# B&R Automation Studio project BenchEDM_AS6 (part 4)

#### HA_Matrix.fun - Exported functions and function blocks
```iecst
FUNCTION HA_Matrix_Tran : BOOL
	VAR_INPUT
		pIn : UDINT;
		pOut : UDINT;
	END_VAR
	VAR
		Internal : HA_Matrix_Internal_typ;
	END_VAR
END_FUNCTION

FUNCTION HA_Matrix_SwapR : BOOL
	VAR_INPUT
		Swap1 : DINT;
		Swap2 : DINT;
		pIn : UDINT;
	END_VAR
	VAR
		Internal : HA_Matrix_Internal_typ;
	END_VAR
END_FUNCTION

FUNCTION HA_Matrix_SwapC : BOOL
	VAR_INPUT
		Swap1 : DINT;
		Swap2 : DINT;
		pIn : UDINT;
	END_VAR
	VAR
		Internal : HA_Matrix_Internal_typ;
	END_VAR
END_FUNCTION

FUNCTION HA_Matrix_Sub : BOOL
	VAR_INPUT
		pIn1 : UDINT;
		pIn2 : UDINT;
		pOut : UDINT;
	END_VAR
	VAR
		Internal : HA_Matrix_Internal_typ;
	END_VAR
END_FUNCTION

FUNCTION HA_Matrix_Rref : BOOL
	VAR_INPUT
		pIn : UDINT;
		pOut : UDINT;
	END_VAR
	VAR
		Internal : HA_Matrix_Internal_typ;
	END_VAR
END_FUNCTION

FUNCTION HA_Matrix_Mult : BOOL
	VAR_INPUT
		pIn1 : UDINT;
		pIn2 : UDINT;
		pOut : UDINT;
	END_VAR
	VAR
		Internal : HA_Matrix_Internal_typ;
	END_VAR
END_FUNCTION

FUNCTION HA_Matrix_Inc : BOOL
	VAR_INPUT
		pIn : UDINT;
	END_VAR
	VAR
		Internal : HA_Matrix_Internal_typ;
	END_VAR
END_FUNCTION

FUNCTION HA_Matrix_I : BOOL
	VAR_INPUT
		pIn : UDINT;
	END_VAR
	VAR
		Internal : HA_Matrix_Internal_typ;
	END_VAR
END_FUNCTION

FUNCTION HA_Matrix_Fill : BOOL
	VAR_INPUT
		FillValue : LREAL;
		pIn : UDINT;
	END_VAR
	VAR
		Internal : HA_Matrix_Internal_typ;
	END_VAR
END_FUNCTION

FUNCTION HA_Matrix_Det : LREAL
	VAR_INPUT
		pIn : UDINT;
		pTemp : UDINT;
		pResult : UDINT;
	END_VAR
	VAR
		Internal : HA_Matrix_Internal_typ;
	END_VAR
END_FUNCTION

FUNCTION HA_Matrix_Add : BOOL
	VAR_INPUT
		pIn1 : UDINT;
		pIn2 : UDINT;
		pOut : UDINT;
	END_VAR
	VAR
		Internal : HA_Matrix_Internal_typ;
	END_VAR
END_FUNCTION

FUNCTION HA_Matrix_Cholesky : BOOL
	VAR_INPUT
		pIn : UDINT;
		pOut : UDINT;
	END_VAR
	VAR
		Internal : HA_Matrix_Internal_typ;
	END_VAR
END_FUNCTION

FUNCTION HA_Matrix_CholSolve : BOOL
	VAR_INPUT
		pL : UDINT;
		pB : UDINT;
		pOut : UDINT;
	END_VAR
	VAR
		Internal : HA_Matrix_Internal_typ;
	END_VAR
END_FUNCTION

FUNCTION HA_Matrix_XtX : BOOL
	VAR_INPUT
		pX : UDINT;
		pOut : UDINT;
	END_VAR
	VAR
		Internal : HA_Matrix_Internal_typ;
	END_VAR
END_FUNCTION

FUNCTION HA_Matrix_XtY : BOOL
	VAR_INPUT
		pX : UDINT;
		pY : UDINT;
		pOut : UDINT;
	END_VAR
	VAR
		Internal : HA_Matrix_Internal_typ;
	END_VAR
END_FUNCTION

FUNCTION HA_Matrix_AddRidge : BOOL
	VAR_INPUT
		pInOut : UDINT;
		Lambda : LREAL;
	END_VAR
	VAR
		Internal : HA_Matrix_Internal_typ;
	END_VAR
END_FUNCTION

FUNCTION HA_Matrix_RLS : BOOL
	VAR_INPUT
		pTheta : UDINT;
		pP : UDINT;
		pX : UDINT;
		Y : LREAL;
		Lambda : LREAL;
		pTemp : UDINT;
	END_VAR
	VAR
		Internal : HA_Matrix_Internal_typ;
	END_VAR
END_FUNCTION

FUNCTION HA_Matrix_RLS_Init : BOOL
	VAR_INPUT
		pTheta : UDINT;
		pP : UDINT;
		InitVariance : LREAL;
	END_VAR
	VAR
		Internal : HA_Matrix_Internal_typ;
	END_VAR
END_FUNCTION

FUNCTION HA_Matrix_Predict : BOOL
	VAR_INPUT
		pX : UDINT;
		pBeta : UDINT;
		pOut : UDINT;
	END_VAR
	VAR
		Internal : HA_Matrix_Internal_typ;
	END_VAR
END_FUNCTION

FUNCTION HA_Matrix_BuildLags : BOOL
	VAR_INPUT
		pY_history : UDINT;
		pU_history : UDINT;
		LagOrder : DINT;
		NumOutputs : DINT;
		NumInputs : DINT;
		pOut : UDINT;
	END_VAR
	VAR
		Internal : HA_Matrix_Internal_typ;
	END_VAR
END_FUNCTION

FUNCTION HA_Matrix_RollingUpdate : BOOL
	VAR_INPUT
		pBuffer : UDINT;
		NewValue : LREAL;
	END_VAR
	VAR
		Internal : HA_Matrix_Internal_typ;
	END_VAR
END_FUNCTION

FUNCTION HA_Matrix_RMSE : LREAL
	VAR_INPUT
		pY_true : UDINT;
		pY_pred : UDINT;
	END_VAR
	VAR
		Internal : HA_Matrix_Internal_typ;
	END_VAR
END_FUNCTION

FUNCTION HA_Matrix_Residuals : BOOL
	VAR_INPUT
		pY_true : UDINT;
		pY_pred : UDINT;
		pOut : UDINT;
	END_VAR
	VAR
		Internal : HA_Matrix_Internal_typ;
	END_VAR
END_FUNCTION

FUNCTION HA_Matrix_R2Score : LREAL
	VAR_INPUT
		pY_true : UDINT;
		pY_pred : UDINT;
	END_VAR
	VAR
		Internal : HA_Matrix_Internal_typ;
	END_VAR
END_FUNCTION

FUNCTION HA_Matrix_Standardize : BOOL
	VAR_INPUT
		pX : UDINT;
		pMean : UDINT;
		pStd : UDINT;
		Mode : DINT;
	END_VAR
	VAR
		Internal : HA_Matrix_Internal_typ;
	END_VAR
END_FUNCTION

FUNCTION HA_Matrix_PolyExpand : BOOL
	VAR_INPUT
		pX : UDINT;
		Order : DINT;
		pOut : UDINT;
	END_VAR
	VAR
		Internal : HA_Matrix_Internal_typ;
	END_VAR
END_FUNCTION

FUNCTION HA_Matrix_Diff : BOOL
	VAR_INPUT
		pX : UDINT;
		pOut : UDINT;
	END_VAR
	VAR
		Internal : HA_Matrix_Internal_typ;
	END_VAR
END_FUNCTION

FUNCTION HA_Matrix_AddBias : BOOL
	VAR_INPUT
		pX : UDINT;
		pOut : UDINT;
	END_VAR
	VAR
		Internal : HA_Matrix_Internal_typ;
	END_VAR
END_FUNCTION

FUNCTION HA_Matrix_PredictMultiStep : BOOL
	VAR_INPUT
		pState : UDINT;
		pBeta : UDINT;
		pHistory : UDINT;
		Steps : DINT;
		LagOrder : DINT;
		PolyOrder : DINT;
		UseDerivative : BOOL;
		UseBias : BOOL;
		pOut : UDINT;
		pLagTemp : UDINT;
		pPolyTemp : UDINT;
		pFeatTemp : UDINT;
		pPredTemp : UDINT;
		pWorkState : UDINT;
		pWorkHist : UDINT;
	END_VAR
	VAR
		Internal : HA_Matrix_Internal_typ;
		Success : BOOL;
	END_VAR
END_FUNCTION

FUNCTION HA_Matrix_Ridge_Fit : BOOL
	VAR_INPUT
		pX : UDINT;
		pY : UDINT;
		Lambda : LREAL;
		UseBias : BOOL;
		WarmupSteps : DINT;
		pBeta : UDINT;
		pXtX : UDINT;
		pXtY : UDINT;
		pL : UDINT;
		pXwork : UDINT;
		pYwork : UDINT;
	END_VAR
	VAR
		Internal : HA_Matrix_Internal_typ;
		Success : BOOL;
	END_VAR
END_FUNCTION

FUNCTION HA_Matrix_BuildLagsStride : BOOL
	VAR_INPUT
		pY_history : UDINT;
		pU_history : UDINT;
		LagOrder : DINT;
		NumOutputs : DINT;
		NumInputs : DINT;
		Stride : DINT;
		pOut : UDINT;
	END_VAR
	VAR
		Internal : HA_Matrix_Internal_typ;
	END_VAR
END_FUNCTION

FUNCTION HA_Matrix_InitStateBuffer : BOOL
	VAR_INPUT
		pX : UDINT;
		LagOrder : DINT;
		pState : UDINT;
		pHistory : UDINT;
	END_VAR
	VAR
		Internal : HA_Matrix_Internal_typ;
	END_VAR
END_FUNCTION

FUNCTION HA_Matrix_NGRC_BuildTrainingData : BOOL
	VAR_INPUT
		pX : UDINT;
		LagOrder : DINT;
		PolyOrder : DINT;
		Stride : DINT;
		UseBias : BOOL;
		WarmupSteps : DINT;
		pOut : UDINT;
		pLagWork : UDINT;
		pPolyWork : UDINT;
	END_VAR
	VAR
		Internal : HA_Matrix_Internal_typ;
		Success : BOOL;
	END_VAR
END_FUNCTION

FUNCTION HA_Matrix_NGRC_Fit : BOOL
	VAR_INPUT
		pX : UDINT;
		pY : UDINT;
		LagOrder : DINT;
		PolyOrder : DINT;
		Stride : DINT;
		Lambda : LREAL;
		UseBias : BOOL;
		UseDerivative : BOOL;
		WarmupSteps : DINT;
		pBeta : UDINT;
		pXtX : UDINT;
		pXtY : UDINT;
		pL : UDINT;
		pLagWork : UDINT;
		pPolyWork : UDINT;
		pFeatWork : UDINT;
		pYwork : UDINT;
	END_VAR
	VAR
		Internal : HA_Matrix_Internal_typ;
		Success : BOOL;
	END_VAR
END_FUNCTION

FUNCTION HA_Matrix_NGRC_InitState : BOOL
	VAR_INPUT
		pX : UDINT;
		LagOrder : DINT;
		Stride : DINT;
		pState : UDINT;
		pHistory : UDINT;
	END_VAR
	VAR
		Internal : HA_Matrix_Internal_typ;
	END_VAR
END_FUNCTION

FUNCTION HA_Matrix_NGRC_Predict : BOOL
	VAR_INPUT
		pHistory : UDINT;
		pBeta : UDINT;
		LagOrder : DINT;
		PolyOrder : DINT;
		UseBias : BOOL;
		pOut : UDINT;
		pLagWork : UDINT;
		pPolyWork : UDINT;
		pFeatWork : UDINT;
	END_VAR
	VAR
		Internal : HA_Matrix_Internal_typ;
		Success : BOOL;
	END_VAR
END_FUNCTION

FUNCTION HA_Matrix_NGRC_PredictMultiStep : BOOL
	VAR_INPUT
		pState : UDINT;
		pBeta : UDINT;
		pHistory : UDINT;
		Steps : DINT;
		LagOrder : DINT;
		PolyOrder : DINT;
		Stride : DINT;
		UseBias : BOOL;
		UseDerivative : BOOL;
		pOut : UDINT;
		pLagWork : UDINT;
		pPolyWork : UDINT;
		pFeatWork : UDINT;
		pPredWork : UDINT;
		pWorkState : UDINT;
		pWorkHist : UDINT;
	END_VAR
	VAR
		Internal : HA_Matrix_Internal_typ;
		Success : BOOL;
	END_VAR
END_FUNCTION

FUNCTION_BLOCK FB_NGRC
	VAR_INPUT
		Enable : BOOL;
		Train : BOOL;
		Predict : BOOL;
		PredictSteps : DINT;
		Reset : BOOL;
	END_VAR
	VAR_OUTPUT
		Status : NGRC_Status_enum;
		Error : NGRC_Error_enum;
		Ready : BOOL;
		Busy : BOOL;
		Done : BOOL;
		Stats : NGRC_Stats_typ;
	END_VAR
	VAR_IN_OUT
		Config : NGRC_Config_typ;
		TrainingData : HA_Matrix_Array_typ;
		PredictionOutput : HA_Matrix_Array_typ;
	END_VAR
	VAR
		Internal : NGRC_Internal_typ;
		TrainTrigger : BOOL;
		PredictTrigger : BOOL;
		ResetTrigger : BOOL;
		Success : BOOL;
		StartTime : UDINT;
		NumDims : DINT;
		NumSamples : DINT;
		IsTrained : BOOL;
	END_VAR
END_FUNCTION_BLOCK

FUNCTION_BLOCK FB_NGRC_Online
	VAR_INPUT
		Enable : BOOL;
		NewSample : BOOL;
		PredictNext : BOOL;
		Reset : BOOL;
	END_VAR
	VAR_OUTPUT
		Status : NGRC_Status_enum;
		Error : NGRC_Error_enum;
		Ready : BOOL;
		PredictionValid : BOOL;
	END_VAR
	VAR_IN_OUT
		Config : NGRC_Config_typ;
		CurrentValue : HA_Matrix_Array_typ;
		Prediction : HA_Matrix_Array_typ;
		TrainedModel : FB_NGRC;
	END_VAR
	VAR
		History : HA_Matrix_Array_typ;
		State : HA_Matrix_Array_typ;
		PredWork : HA_Matrix_Array_typ;
		NewSampleTrigger : BOOL;
		PredictTrigger : BOOL;
		Success : BOOL;
		Initialized : BOOL;
		NumDims : DINT;
		i : DINT;
		temp : LREAL;
	END_VAR
END_FUNCTION_BLOCK

FUNCTION_BLOCK FB_NGRC_Simple
	VAR_INPUT
		Execute : BOOL;
		LagOrder : DINT;
		PolyOrder : DINT;
		Stride : DINT;
		Lambda : LREAL;
		PredictSteps : DINT;
	END_VAR
	VAR_OUTPUT
		Done : BOOL;
		Busy : BOOL;
		Error : BOOL;
		ErrorID : NGRC_Error_enum;
	END_VAR
	VAR_IN_OUT
		TrainingData : HA_Matrix_Array_typ;
		Predictions : HA_Matrix_Array_typ;
	END_VAR
	VAR
		Model : FB_NGRC;
		InternalConfig : NGRC_Config_typ;
		InternalTrainData : HA_Matrix_Array_typ;
		InternalPredictions : HA_Matrix_Array_typ;
		ExecuteTrigger : BOOL;
		State : DINT;
	END_VAR
END_FUNCTION_BLOCK

FUNCTION_BLOCK FB_NGRC_Continuous
	VAR_INPUT
		Enable : BOOL;
		Reset : BOOL;
		NewSample : LREAL;
	END_VAR
	VAR_OUTPUT
		PredictedNext : LREAL;
		Predicted5Step : ARRAY[0..4] OF LREAL;
		Status : NGRC_Continuous_Status_typ;
		Metrics : NGRC_Continuous_Metrics_typ;
	END_VAR
	VAR_IN_OUT
		Config : NGRC_Continuous_Config_typ;
	END_VAR
	VAR
		Model_Active : FB_NGRC;
		Model_Training : FB_NGRC;
		Predictor_Online : FB_NGRC_Online;
		DataBuffer : ARRAY[0..499] OF LREAL;
		BufferIndex : DINT := 0;
		BufferFull : BOOL := FALSE;
		TrainingData : HA_Matrix_Array_typ;
		CurrentSample : HA_Matrix_Array_typ;
		PredictionBuffer : HA_Matrix_Array_typ;
		PredictionOutput_Active : HA_Matrix_Array_typ;
		PredictionOutput_Training : HA_Matrix_Array_typ;
		TrainingState : DINT := 0;
		StateFlags : StateFlags_typ;
		ModelSwapReady : BOOL := FALSE;
		SamplesSinceRetrain : DINT := 0;
		RetrainTrigger : BOOL := FALSE;
		PredictionState : DINT := 0;
		MultiStepState : DINT := 0;
		ErrorSum_1Step : LREAL := 0.0;
		ErrorCount_1Step : DINT := 0;
		MaxError_1Step : LREAL := 0.0;
		LastPrediction : LREAL := 0.0;
		ErrorSum_5Step : LREAL := 0.0;
		ErrorCount_5Step : DINT := 0;
		ErrorWindow : ARRAY[0..19] OF LREAL;
		ErrorWindowIndex : DINT := 0;
		PredictionHistory : ARRAY[0..4] OF LREAL;
		PredictionAge : ARRAY[0..4] OF DINT;
		i : DINT;
		j : DINT;
		temp : LREAL;
		CycleCount : DINT := 0;
	END_VAR
END_FUNCTION_BLOCK

FUNCTION_BLOCK FB_NGRC_Continuous_MultiVar
VAR_INPUT
	Enable : BOOL;
	Reset : BOOL;
	NewSample : ARRAY[0..9] OF LREAL;
END_VAR
VAR_OUTPUT
	PredictedNext : ARRAY[0..9] OF LREAL;
	Predicted5Step : ARRAY[0..9, 0..4] OF LREAL;
	Status : NGRC_MultiVar_Status_typ;
	Metrics : NGRC_MultiVar_Metrics_typ;
END_VAR
VAR_IN_OUT
	Config : NGRC_MultiVar_Config_typ;
END_VAR
VAR
	Model_Active : FB_NGRC;
	Model_Training : FB_NGRC;
	Predictor_Online : FB_NGRC_Online;
	DataBuffer : ARRAY[0..4999] OF LREAL;
	BufferIndex : DINT := 0;
	BufferFull : BOOL := FALSE;
	TrainingData : HA_Matrix_Array_typ;
	CurrentSample : HA_Matrix_Array_typ;
	PredictionBuffer : HA_Matrix_Array_typ;
	PredictionOutput_Active : HA_Matrix_Array_typ;
	PredictionOutput_Training : HA_Matrix_Array_typ;
	StateFlags : StateFlags_typ;
	TrainingState : DINT := 0;
	ModelSwapReady : BOOL := FALSE;
	SamplesSinceRetrain : DINT := 0;
	RetrainTrigger : BOOL := FALSE;
	PredictionState : DINT := 0;
	MultiStepState : DINT := 0;
	ErrorSum_1Step : ARRAY[0..9] OF LREAL;
	ErrorCount_1Step : ARRAY[0..9] OF DINT;
	MaxError_1Step : ARRAY[0..9] OF LREAL;
	LastPrediction : ARRAY[0..9] OF LREAL;
	ErrorSum_5Step : ARRAY[0..9] OF LREAL;
	ErrorCount_5Step : ARRAY[0..9] OF DINT;
	ErrorWindow : ARRAY[0..19] OF LREAL;
	ErrorWindowIndex : DINT := 0;
	TotalErrorSum : LREAL := 0.0;
	TotalErrorCount : DINT := 0;
	PredictionHistory : ARRAY[0..9, 0..4] OF LREAL;
	PredictionAge : ARRAY[0..9, 0..4] OF DINT;
	i : DINT;
	j : DINT;
	k : DINT;
	temp : LREAL;
	tempSum : LREAL;
	CycleCount : DINT := 0;
	NumVars : DINT;
	BufferOffset : DINT;
END_VAR
END_FUNCTION_BLOCK
```

#### HA_Matrix_Tran.st
```iecst
(* Transpose *)
FUNCTION HA_Matrix_Tran
	HA_Matrix_Tran		 			:= TRUE;
	brsmemset(ADR(Internal),0,SIZEOF(Internal));
	Internal.sizeArray				:= SIZEOF(LREAL)*(MAX_HA_MATRIX_ARRAY_IDX+1);
	Internal.sizeTotal				:= Internal.sizeArray + SIZEOF(DINT)*2;
	brsmemcpy(ADR(Internal.row1),pIn+Internal.sizeArray,4);
	brsmemcpy(ADR(Internal.col1),pIn+Internal.sizeArray+4,4);
	Internal.row2					:= Internal.col1;
	Internal.col2					:= Internal.row1;
	IF pIn = 0 OR pOut = 0 OR Internal.row1 = 0 OR Internal.col1 = 0 OR Internal.row1*Internal.col1 > MAX_HA_MATRIX_ARRAY_IDX+1 THEN
		HA_Matrix_Tran	 			:= FALSE;
	ELSE
		brsmemset(pOut,0,Internal.sizeTotal);
		brsmemcpy(pOut+Internal.sizeArray,ADR(Internal.row2),4);
		brsmemcpy(pOut+Internal.sizeArray+4,ADR(Internal.col2),4);
		FOR Internal.i1 := 0 TO (Internal.row1*Internal.col1)-1 DO
			brsmemcpy(pOut+(((Internal.i1 MOD Internal.col1)*Internal.row1)+Internal.i1/Internal.col1)*8,pIn+Internal.i1*8,8);
		END_FOR;
	END_IF;
END_FUNCTION
```

#### HA_Matrix_Mult.st
```iecst
(* Multiply *)
FUNCTION HA_Matrix_Mult
	HA_Matrix_Mult 					:= TRUE;
	brsmemset(ADR(Internal),0,SIZEOF(Internal));
	Internal.sizeArray				:= SIZEOF(LREAL)*(MAX_HA_MATRIX_ARRAY_IDX+1);
	Internal.sizeTotal				:= Internal.sizeArray + SIZEOF(DINT)*2;
	brsmemcpy(ADR(Internal.row1),pIn1+Internal.sizeArray,4);
	brsmemcpy(ADR(Internal.col1),pIn1+Internal.sizeArray+4,4);
	brsmemcpy(ADR(Internal.row2),pIn2+Internal.sizeArray,4);
	brsmemcpy(ADR(Internal.col2),pIn2+Internal.sizeArray+4,4);
	IF pIn1 = 0 OR pIn2 = 0 OR pOut = 0 OR Internal.row1 = 0 OR Internal.col1 = 0 OR Internal.row2 = 0 OR Internal.col2 = 0 OR Internal.row1*Internal.col1 > MAX_HA_MATRIX_ARRAY_IDX+1 OR Internal.row2*Internal.col2 > MAX_HA_MATRIX_ARRAY_IDX+1 OR Internal.row1*Internal.col2 > MAX_HA_MATRIX_ARRAY_IDX+1 OR Internal.col1 <> Internal.row2 THEN
		HA_Matrix_Mult	 			:= FALSE;
	ELSE
		brsmemset(pOut,0,Internal.sizeTotal);
		brsmemcpy(pOut+Internal.sizeArray,ADR(Internal.row1),4);
		brsmemcpy(pOut+Internal.sizeArray+4,ADR(Internal.col2),4);
		FOR Internal.i1 := 0 TO Internal.row1-1 DO
		    FOR Internal.i2 := 0 TO Internal.col2-1 DO
		        Internal.result 	:= 0.0;
		        FOR Internal.i3 := 0 TO Internal.col1-1 DO
					brsmemcpy(ADR(Internal.temp1),pIn1+(Internal.i1*Internal.col1+Internal.i3)*8,8);
					brsmemcpy(ADR(Internal.temp2),pIn2+(Internal.i3*Internal.col2+Internal.i2)*8,8);
		            Internal.result := Internal.result + Internal.temp1 * Internal.temp2;
		        END_FOR;
				brsmemcpy(pOut+(Internal.i1*Internal.col2+Internal.i2)*8,ADR(Internal.result),8);
		    END_FOR;
		END_FOR;
	END_IF;
END_FUNCTION
```

#### HA_Matrix_Add.st
```iecst
(* Addition *)
FUNCTION HA_Matrix_Add
	HA_Matrix_Add	 				:= TRUE;
	brsmemset(ADR(Internal),0,SIZEOF(Internal));
	Internal.sizeArray				:= SIZEOF(LREAL)*(MAX_HA_MATRIX_ARRAY_IDX+1);
	Internal.sizeTotal				:= Internal.sizeArray + SIZEOF(DINT)*2;
	brsmemcpy(ADR(Internal.row1),pIn1+Internal.sizeArray,4);
	brsmemcpy(ADR(Internal.col1),pIn1+Internal.sizeArray+4,4);
	brsmemcpy(ADR(Internal.row2),pIn2+Internal.sizeArray,4);
	brsmemcpy(ADR(Internal.col2),pIn2+Internal.sizeArray+4,4);
	IF pIn1 = 0 OR pIn2 = 0 OR pOut = 0 OR Internal.row1 = 0 OR Internal.col1 = 0 OR Internal.row2 = 0 OR Internal.col2 = 0 OR Internal.row1*Internal.col1 > MAX_HA_MATRIX_ARRAY_IDX+1 OR Internal.row2*Internal.col2 > MAX_HA_MATRIX_ARRAY_IDX+1 OR Internal.row1 <> Internal.row2 OR Internal.col1 <> Internal.col2 THEN
		HA_Matrix_Add	 			:= FALSE;
	ELSE
		brsmemset(pOut,0,Internal.sizeTotal);
		brsmemcpy(pOut+Internal.sizeArray,ADR(Internal.row1),4);
		brsmemcpy(pOut+Internal.sizeArray+4,ADR(Internal.col1),4);
		FOR Internal.i1 := 0 TO Internal.row1-1 DO
		    FOR Internal.i2 := 0 TO Internal.col1-1 DO
				brsmemcpy(ADR(Internal.temp1),pIn1+(Internal.i1*Internal.col1+Internal.i2)*8,8);
				brsmemcpy(ADR(Internal.temp2),pIn2+(Internal.i1*Internal.col1+Internal.i2)*8,8);
		        Internal.result 	:= Internal.temp1 + Internal.temp2;
				brsmemcpy(pOut+(Internal.i1*Internal.col1+Internal.i2)*8,ADR(Internal.result),8);
		    END_FOR;
		END_FOR;
	END_IF;
END_FUNCTION
```

#### HA_Matrix_Sub.st
```iecst
(* Subtraction *)
FUNCTION HA_Matrix_Sub
	HA_Matrix_Sub		 			:= TRUE;
	brsmemset(ADR(Internal),0,SIZEOF(Internal));
	Internal.sizeArray				:= SIZEOF(LREAL)*(MAX_HA_MATRIX_ARRAY_IDX+1);
	Internal.sizeTotal				:= Internal.sizeArray + SIZEOF(DINT)*2;
	brsmemcpy(ADR(Internal.row1),pIn1+Internal.sizeArray,4);
	brsmemcpy(ADR(Internal.col1),pIn1+Internal.sizeArray+4,4);
	brsmemcpy(ADR(Internal.row2),pIn2+Internal.sizeArray,4);
	brsmemcpy(ADR(Internal.col2),pIn2+Internal.sizeArray+4,4);
	IF pIn1 = 0 OR pIn2 = 0 OR pOut = 0 OR Internal.row1 = 0 OR Internal.col1 = 0 OR Internal.row2 = 0 OR Internal.col2 = 0 OR Internal.row1*Internal.col1 > MAX_HA_MATRIX_ARRAY_IDX+1 OR Internal.row2*Internal.col2 > MAX_HA_MATRIX_ARRAY_IDX+1 OR Internal.row1 <> Internal.row2 OR Internal.col1 <> Internal.col2 THEN
		HA_Matrix_Sub	 			:= FALSE;
	ELSE
		brsmemset(pOut,0,Internal.sizeTotal);
		brsmemcpy(pOut+Internal.sizeArray,ADR(Internal.row1),4);
		brsmemcpy(pOut+Internal.sizeArray+4,ADR(Internal.col1),4);
		FOR Internal.i1 := 0 TO Internal.row1-1 DO
		    FOR Internal.i2 := 0 TO Internal.col1-1 DO
				brsmemcpy(ADR(Internal.temp1),pIn1+(Internal.i1*Internal.col1+Internal.i2)*8,8);
				brsmemcpy(ADR(Internal.temp2),pIn2+(Internal.i1*Internal.col1+Internal.i2)*8,8);
		        Internal.result 	:= Internal.temp1 - Internal.temp2;
				brsmemcpy(pOut+(Internal.i1*Internal.col1+Internal.i2)*8,ADR(Internal.result),8);
		    END_FOR;
		END_FOR;
	END_IF;
END_FUNCTION
```

#### HA_Matrix_Fill.st
```iecst
(* Fill *)
FUNCTION HA_Matrix_Fill
	HA_Matrix_Fill	 				:= TRUE;
	brsmemset(ADR(Internal),0,SIZEOF(Internal));
	Internal.sizeArray				:= SIZEOF(LREAL)*(MAX_HA_MATRIX_ARRAY_IDX+1);
	Internal.sizeTotal				:= Internal.sizeArray + SIZEOF(DINT)*2;
	brsmemcpy(ADR(Internal.row1),pIn+Internal.sizeArray,4);
	brsmemcpy(ADR(Internal.col1),pIn+Internal.sizeArray+4,4);
	IF pIn = 0 OR Internal.row1 = 0 OR Internal.col1 = 0 OR Internal.row1*Internal.col1 > MAX_HA_MATRIX_ARRAY_IDX+1 THEN
		HA_Matrix_Fill	 			:= FALSE;
	ELSE
		FOR Internal.i1 := 0 TO Internal.row1-1 DO
		    FOR Internal.i2 := 0 TO Internal.col1-1 DO
				brsmemcpy(pIn+(Internal.i1*Internal.col1+Internal.i2)*8,ADR(FillValue),8);
		    END_FOR;
		END_FOR;
	END_IF;
END_FUNCTION
```

#### HA_Matrix_Inc.st
```iecst
(* Fill Incrementing *)
FUNCTION HA_Matrix_Inc
	HA_Matrix_Inc	 				:= TRUE;
	brsmemset(ADR(Internal),0,SIZEOF(Internal));
	Internal.sizeArray				:= SIZEOF(LREAL)*(MAX_HA_MATRIX_ARRAY_IDX+1);
	Internal.sizeTotal				:= Internal.sizeArray + SIZEOF(DINT)*2;
	brsmemcpy(ADR(Internal.row1),pIn+Internal.sizeArray,4);
	brsmemcpy(ADR(Internal.col1),pIn+Internal.sizeArray+4,4);
	IF pIn = 0 OR Internal.row1 = 0 OR Internal.col1 = 0 OR Internal.row1*Internal.col1 > MAX_HA_MATRIX_ARRAY_IDX+1 THEN
		HA_Matrix_Inc	 			:= FALSE;
	ELSE
		FOR Internal.i1 := 0 TO Internal.row1-1 DO
		    FOR Internal.i2 := 0 TO Internal.col1-1 DO
				Internal.temp1 		:= DINT_TO_LREAL(Internal.i1*Internal.col1+Internal.i2);
				brsmemcpy(pIn+(Internal.i1*Internal.col1+Internal.i2)*8,ADR(Internal.temp1),8);
		    END_FOR;
		END_FOR;
	END_IF;
END_FUNCTION
```

#### HA_Matrix_I.st
```iecst
(* Identity *)
FUNCTION HA_Matrix_I
	HA_Matrix_I	 					:= TRUE;
	brsmemset(ADR(Internal),0,SIZEOF(Internal));
	Internal.sizeArray				:= SIZEOF(LREAL)*(MAX_HA_MATRIX_ARRAY_IDX+1);
	Internal.sizeTotal				:= Internal.sizeArray + SIZEOF(DINT)*2;
	brsmemcpy(ADR(Internal.row1),pIn+Internal.sizeArray,4);
	brsmemcpy(ADR(Internal.col1),pIn+Internal.sizeArray+4,4);
	IF pIn = 0 OR Internal.row1 = 0 OR Internal.col1 = 0 OR Internal.row1*Internal.col1 > MAX_HA_MATRIX_ARRAY_IDX+1 OR Internal.row1 <> Internal.col1 THEN
		HA_Matrix_I	 				:= FALSE;
	ELSE
		FOR Internal.i1 := 0 TO Internal.row1-1 DO
		    FOR Internal.i2 := 0 TO Internal.col1-1 DO
				Internal.temp1 		:= 0.0;
				IF Internal.i1 = Internal.i2 THEN
					Internal.temp1 	:= 1.0;
				END_IF;
				brsmemcpy(pIn+(Internal.i1*Internal.row1+Internal.i2)*8,ADR(Internal.temp1),8);
		    END_FOR;
		END_FOR;
	END_IF;
END_FUNCTION
```

#### HA_Matrix_SwapR.st
```iecst
(* Swap Row *)
FUNCTION HA_Matrix_SwapR
	HA_Matrix_SwapR	 				:= TRUE;
	brsmemset(ADR(Internal),0,SIZEOF(Internal));
	Internal.sizeArray				:= SIZEOF(LREAL)*(MAX_HA_MATRIX_ARRAY_IDX+1);
	Internal.sizeTotal				:= Internal.sizeArray + SIZEOF(DINT)*2;
	brsmemcpy(ADR(Internal.row1),pIn+Internal.sizeArray,4);
	brsmemcpy(ADR(Internal.col1),pIn+Internal.sizeArray+4,4);
	IF pIn = 0 OR Internal.row1 = 0 OR Internal.col1 = 0 OR Internal.row1*Internal.col1 > MAX_HA_MATRIX_ARRAY_IDX+1 OR Swap1 = Swap2 OR Internal.row1-1 < Swap1 OR Internal.row1-1 < Swap2 THEN
		HA_Matrix_SwapR	 			:= FALSE;
	ELSE
		FOR Internal.i1 := 0 TO Internal.col1-1 DO
			brsmemcpy(ADR(Internal.temp1),pIn+(Swap1*Internal.col1+Internal.i1)*8,8);
			brsmemcpy(ADR(Internal.temp2),pIn+(Swap2*Internal.col1+Internal.i1)*8,8);
			brsmemcpy(pIn+(Swap1*Internal.col1+Internal.i1)*8,ADR(Internal.temp2),8);
			brsmemcpy(pIn+(Swap2*Internal.col1+Internal.i1)*8,ADR(Internal.temp1),8);
		END_FOR;
	END_IF;
END_FUNCTION
```

#### HA_Matrix_SwapC.st
```iecst
(* Swap Column *)
FUNCTION HA_Matrix_SwapC
	HA_Matrix_SwapC	 				:= TRUE;
	brsmemset(ADR(Internal),0,SIZEOF(Internal));
	Internal.sizeArray				:= SIZEOF(LREAL)*(MAX_HA_MATRIX_ARRAY_IDX+1);
	Internal.sizeTotal				:= Internal.sizeArray + SIZEOF(DINT)*2;
	brsmemcpy(ADR(Internal.row1),pIn+Internal.sizeArray,4);
	brsmemcpy(ADR(Internal.col1),pIn+Internal.sizeArray+4,4);
	IF pIn = 0 OR Internal.row1 = 0 OR Internal.col1 = 0 OR Internal.row1*Internal.col1 > MAX_HA_MATRIX_ARRAY_IDX+1 OR Swap1 = Swap2 OR Internal.col1-1 < Swap1 OR Internal.col1-1 < Swap2 THEN
		HA_Matrix_SwapC	 			:= FALSE;
	ELSE
		FOR Internal.i1 := 0 TO Internal.row1-1 DO
			brsmemcpy(ADR(Internal.temp1),pIn+(Internal.i1*Internal.col1+Swap1)*8,8);
			brsmemcpy(ADR(Internal.temp2),pIn+(Internal.i1*Internal.col1+Swap2)*8,8);
			brsmemcpy(pIn+(Internal.i1*Internal.col1+Swap1)*8,ADR(Internal.temp2),8);
			brsmemcpy(pIn+(Internal.i1*Internal.col1+Swap2)*8,ADR(Internal.temp1),8);
		END_FOR;
	END_IF;
END_FUNCTION
```

#### HA_Matrix_Det.st
```iecst
(* Determinant *)
FUNCTION HA_Matrix_Det

    HA_Matrix_Det := FALSE;
    brsmemset(ADR(Internal),0,SIZEOF(Internal));
    Internal.sizeArray := SIZEOF(LREAL)*(MAX_HA_MATRIX_ARRAY_IDX+1);
    Internal.sizeTotal := Internal.sizeArray + SIZEOF(DINT)*2;
    brsmemcpy(ADR(Internal.row1),pIn+Internal.sizeArray,4);
    brsmemcpy(ADR(Internal.col1),pIn+Internal.sizeArray+4,4);
    IF pIn = 0 OR pTemp = 0 OR pResult = 0 OR Internal.row1 = 0 OR Internal.col1 = 0 OR Internal.row1 <> Internal.col1 OR Internal.row1*Internal.col1 > MAX_HA_MATRIX_ARRAY_IDX+1 THEN
        Internal.result := 0.0;
        brsmemcpy(pResult,ADR(Internal.result),8);
        HA_Matrix_Det := FALSE;
    ELSE
        IF Internal.row1 = 1 THEN
            brsmemcpy(ADR(Internal.result),pIn,8);
            brsmemcpy(pResult,ADR(Internal.result),8);
            HA_Matrix_Det := TRUE;
        ELSIF Internal.row1 = 2 THEN
            brsmemcpy(ADR(Internal.temp1),pIn+0*8,8);
            brsmemcpy(ADR(Internal.temp2),pIn+1*8,8);
            brsmemcpy(ADR(Internal.temp3),pIn+2*8,8);
            brsmemcpy(ADR(Internal.temp4),pIn+3*8,8);
            Internal.result := Internal.temp1*Internal.temp4 - Internal.temp2*Internal.temp3;
            brsmemcpy(pResult,ADR(Internal.result),8);
            HA_Matrix_Det := TRUE;
        ELSE
            Internal.result := 1.0;  (* Use result to track sign *)
            brsmemcpy(pTemp,pIn,Internal.sizeArray);
            brsmemcpy(pTemp+Internal.sizeArray,pIn+Internal.sizeArray,8);
            FOR Internal.i1 := 0 TO Internal.row1-2 DO
                brsmemcpy(ADR(Internal.temp1),pTemp+(Internal.i1*Internal.col1+Internal.i1)*8,8);
                IF ABS(Internal.temp1) < 1.0e-10 THEN
                    FOR Internal.i2 := Internal.i1+1 TO Internal.row1-1 DO
                        brsmemcpy(ADR(Internal.temp1),pTemp+(Internal.i2*Internal.col1+Internal.i1)*8,8);
                        IF ABS(Internal.temp1) > 1.0e-10 THEN
                            FOR Internal.i3 := 0 TO Internal.col1-1 DO
                                brsmemcpy(ADR(Internal.temp2),pTemp+(Internal.i1*Internal.col1+Internal.i3)*8,8);
                                brsmemcpy(ADR(Internal.temp3),pTemp+(Internal.i2*Internal.col1+Internal.i3)*8,8);
                                brsmemcpy(pTemp+(Internal.i1*Internal.col1+Internal.i3)*8,ADR(Internal.temp3),8);
                                brsmemcpy(pTemp+(Internal.i2*Internal.col1+Internal.i3)*8,ADR(Internal.temp2),8);
                            END_FOR;
                            Internal.result := -Internal.result;  (* Negate sign *)
                            EXIT;
                        END_IF;
                    END_FOR;
                END_IF;
                brsmemcpy(ADR(Internal.temp1),pTemp+(Internal.i1*Internal.col1+Internal.i1)*8,8);
                IF ABS(Internal.temp1) < 1.0e-10 THEN
                    Internal.result := 0.0;
                    brsmemcpy(pResult,ADR(Internal.result),8);
                    HA_Matrix_Det := TRUE;  (* Successfully determined matrix is singular *)
                    RETURN;
                END_IF;
                FOR Internal.i2 := Internal.i1+1 TO Internal.row1-1 DO
                    brsmemcpy(ADR(Internal.temp2),pTemp+(Internal.i2*Internal.col1+Internal.i1)*8,8);
                    Internal.temp3 := Internal.temp2/Internal.temp1;
                    FOR Internal.i3 := Internal.i1 TO Internal.col1-1 DO
                        brsmemcpy(ADR(Internal.temp2),pTemp+(Internal.i2*Internal.col1+Internal.i3)*8,8);
                        brsmemcpy(ADR(Internal.temp4),pTemp+(Internal.i1*Internal.col1+Internal.i3)*8,8);
                        Internal.temp2 := Internal.temp2 - Internal.temp3*Internal.temp4;
                        brsmemcpy(pTemp+(Internal.i2*Internal.col1+Internal.i3)*8,ADR(Internal.temp2),8);
                    END_FOR;
                END_FOR;
            END_FOR;
            (* result already contains the sign, now multiply by diagonal elements *)
            FOR Internal.i1 := 0 TO Internal.row1-1 DO
                brsmemcpy(ADR(Internal.temp1),pTemp+(Internal.i1*Internal.col1+Internal.i1)*8,8);
                Internal.result := Internal.result*Internal.temp1;
            END_FOR;
            brsmemcpy(pResult,ADR(Internal.result),8);
            HA_Matrix_Det := TRUE;
        END_IF;
    END_IF;
END_FUNCTION
```

#### HA_Matrix_Rref.st
```iecst
(* Reduced Row Echelon Form *)
FUNCTION HA_Matrix_Rref
	HA_Matrix_Rref		 			:= TRUE;
	brsmemset(ADR(Internal),0,SIZEOF(Internal));
	Internal.sizeArray				:= SIZEOF(LREAL)*(MAX_HA_MATRIX_ARRAY_IDX+1);
	Internal.sizeTotal				:= Internal.sizeArray + SIZEOF(DINT)*2;
	brsmemcpy(ADR(Internal.row1),pIn+Internal.sizeArray,4);
	brsmemcpy(ADR(Internal.col1),pIn+Internal.sizeArray+4,4);
	IF pIn = 0 OR pOut = 0 OR Internal.row1 = 0 OR Internal.col1 = 0 OR Internal.row1*Internal.col1 > MAX_HA_MATRIX_ARRAY_IDX+1 THEN
		HA_Matrix_Rref	 			:= FALSE;
		brsmemset(pOut,0,Internal.sizeTotal);
		Internal.result				:= 0.0;
		IF pOut <> 0 THEN
			brsmemcpy(pOut,ADR(Internal.row1),4);
		END_IF;
	ELSE
	    brsmemcpy(pOut,pIn,Internal.sizeTotal);
        FOR Internal.i1 := 0 TO Internal.row1-1 DO
			brsmemcpy(ADR(Internal.temp1),pOut+(Internal.i1*Internal.col1+Internal.i1)*8,8);
			IF ABS(Internal.temp1) < 1.0e-10 THEN
        		FOR Internal.i2 := Internal.i1+1 TO Internal.row1-1 DO
					brsmemcpy(ADR(Internal.temp1),pOut+(Internal.i2*Internal.col1+Internal.i1)*8,8);
					IF ABS(Internal.temp1) > 1.0e-10 THEN
						FOR Internal.i3 := 0 TO Internal.col1-1 DO
							brsmemcpy(ADR(Internal.temp2),pOut+(Internal.i1*Internal.col1+Internal.i3)*8,8);
							brsmemcpy(ADR(Internal.temp3),pOut+(Internal.i2*Internal.col1+Internal.i3)*8,8);
							brsmemcpy(pOut+(Internal.i1*Internal.col1+Internal.i3)*8,ADR(Internal.temp3),8);
							brsmemcpy(pOut+(Internal.i2*Internal.col1+Internal.i3)*8,ADR(Internal.temp2),8);
						END_FOR;
						EXIT;
					END_IF;
				END_FOR;
			END_IF;
			brsmemcpy(ADR(Internal.temp1),pOut+(Internal.i1*Internal.col1+Internal.i1)*8,8);
			IF ABS(Internal.temp1) > 1.0e-10 THEN
	            FOR Internal.i2 := 0 TO Internal.col1-1 DO
					brsmemcpy(ADR(Internal.temp2),pOut+(Internal.i1*Internal.col1+Internal.i2)*8,8);
	                Internal.temp3 := Internal.temp2 / Internal.temp1;
					brsmemcpy(pOut+(Internal.i1*Internal.col1+Internal.i2)*8,ADR(Internal.temp3),8);
	            END_FOR;
	            FOR Internal.i2 := 0 TO Internal.row1-1 DO
	                IF Internal.i2 <> Internal.i1 THEN
						brsmemcpy(ADR(Internal.temp1),pOut+(Internal.i2*Internal.col1+Internal.i1)*8,8);
	                    FOR Internal.i3 := 0 TO Internal.col1-1 DO
							brsmemcpy(ADR(Internal.temp2),pOut+(Internal.i2*Internal.col1+Internal.i3)*8,8);
							brsmemcpy(ADR(Internal.temp3),pOut+(Internal.i1*Internal.col1+Internal.i3)*8,8);
							Internal.temp4 := Internal.temp2 - Internal.temp1 * Internal.temp3;
							IF ABS(Internal.temp4) < 1.0e-10 THEN
								Internal.temp4 := 0.0;
							END_IF;
							brsmemcpy(pOut+(Internal.i2*Internal.col1+Internal.i3)*8,ADR(Internal.temp4),8);
	                    END_FOR;
	                END_IF;
	            END_FOR;
			END_IF;
        END_FOR;
		Internal.i3 := 0;
        FOR Internal.i1 := 0 TO Internal.row1-1 DO
			Internal.i4 := 0;
	    	FOR Internal.i2 := 0 TO Internal.col1-1 DO
				brsmemcpy(ADR(Internal.temp1),pOut+(Internal.i1*Internal.col1+Internal.i2)*8,8);
				IF ABS(Internal.temp1) > 1.0e-10 THEN
					Internal.i4 := 1;
				END_IF;
			END_FOR;
			IF Internal.i4 = 0 THEN
				Internal.i3 := Internal.i3 + 1;
			END_IF;
        END_FOR;
		IF pOut <> 0 THEN
			brsmemcpy(pOut,ADR(Internal.i3),4);
		END_IF;
	END_IF;
END_FUNCTION
```

#### HA_Matrix_Cholesky.st
```iecst
(* Cholesky Decomposition *)
FUNCTION HA_Matrix_Cholesky
	HA_Matrix_Cholesky	 			:= TRUE;
	brsmemset(ADR(Internal),0,SIZEOF(Internal));
	Internal.sizeArray				:= SIZEOF(LREAL)*(MAX_HA_MATRIX_ARRAY_IDX+1);
	Internal.sizeTotal				:= Internal.sizeArray + SIZEOF(DINT)*2;
	brsmemcpy(ADR(Internal.row1),pIn+Internal.sizeArray,4);
	brsmemcpy(ADR(Internal.col1),pIn+Internal.sizeArray+4,4);
	IF pIn = 0 OR pOut = 0 OR Internal.row1 = 0 OR Internal.col1 = 0 OR Internal.row1 <> Internal.col1 OR Internal.row1*Internal.col1 > MAX_HA_MATRIX_ARRAY_IDX+1 THEN
		HA_Matrix_Cholesky	 		:= FALSE;
	ELSE
		brsmemset(pOut,0,Internal.sizeTotal);
		brsmemcpy(pOut+Internal.sizeArray,ADR(Internal.row1),4);
		brsmemcpy(pOut+Internal.sizeArray+4,ADR(Internal.col1),4);
		FOR Internal.i1 := 0 TO Internal.row1-1 DO
		    FOR Internal.i2 := 0 TO Internal.i1 DO
				Internal.result 	:= 0.0;
		        IF Internal.i1 = Internal.i2 THEN
		            FOR Internal.i3 := 0 TO Internal.i2-1 DO
						brsmemcpy(ADR(Internal.temp1),pOut+(Internal.i1*Internal.col1+Internal.i3)*8,8);
		                Internal.result := Internal.result + Internal.temp1*Internal.temp1;
		            END_FOR;
					brsmemcpy(ADR(Internal.temp1),pIn+(Internal.i1*Internal.col1+Internal.i1)*8,8);
		            Internal.result := Internal.temp1 - Internal.result;
		            IF Internal.result < 1.0e-10 THEN
		                HA_Matrix_Cholesky := FALSE;
		                RETURN;
		            END_IF;
		            Internal.result := SQRT(Internal.result);
					brsmemcpy(pOut+(Internal.i1*Internal.col1+Internal.i1)*8,ADR(Internal.result),8);
		        ELSE
		            FOR Internal.i3 := 0 TO Internal.i2-1 DO
						brsmemcpy(ADR(Internal.temp1),pOut+(Internal.i1*Internal.col1+Internal.i3)*8,8);
						brsmemcpy(ADR(Internal.temp2),pOut+(Internal.i2*Internal.col1+Internal.i3)*8,8);
		                Internal.result := Internal.result + Internal.temp1*Internal.temp2;
		            END_FOR;
					brsmemcpy(ADR(Internal.temp1),pIn+(Internal.i1*Internal.col1+Internal.i2)*8,8);
					brsmemcpy(ADR(Internal.temp2),pOut+(Internal.i2*Internal.col1+Internal.i2)*8,8);
		            Internal.result := (Internal.temp1 - Internal.result)/Internal.temp2;
					brsmemcpy(pOut+(Internal.i1*Internal.col1+Internal.i2)*8,ADR(Internal.result),8);
		        END_IF;
		    END_FOR;
		END_FOR;
	END_IF;
END_FUNCTION
```

#### HA_Matrix_CholSolve.st
```iecst
(* Cholesky Solve *)
FUNCTION HA_Matrix_CholSolve
	HA_Matrix_CholSolve	 			:= TRUE;
	brsmemset(ADR(Internal),0,SIZEOF(Internal));
	Internal.sizeArray				:= SIZEOF(LREAL)*(MAX_HA_MATRIX_ARRAY_IDX+1);
	Internal.sizeTotal				:= Internal.sizeArray + SIZEOF(DINT)*2;
	brsmemcpy(ADR(Internal.row1),pL+Internal.sizeArray,4);
	brsmemcpy(ADR(Internal.col1),pL+Internal.sizeArray+4,4);
	brsmemcpy(ADR(Internal.row2),pB+Internal.sizeArray,4);
	brsmemcpy(ADR(Internal.col2),pB+Internal.sizeArray+4,4);
	IF pL = 0 OR pB = 0 OR pOut = 0 OR Internal.row1 = 0 OR Internal.col1 = 0 OR Internal.row2 = 0 OR Internal.col2 = 0 OR Internal.row1 <> Internal.col1 OR Internal.row1 <> Internal.row2 OR Internal.row1*Internal.col1 > MAX_HA_MATRIX_ARRAY_IDX+1 OR Internal.row2*Internal.col2 > MAX_HA_MATRIX_ARRAY_IDX+1 THEN
		HA_Matrix_CholSolve	 		:= FALSE;
	ELSE
		brsmemset(pOut,0,Internal.sizeTotal);
		brsmemcpy(pOut+Internal.sizeArray,ADR(Internal.row2),4);
		brsmemcpy(pOut+Internal.sizeArray+4,ADR(Internal.col2),4);
		FOR Internal.i3 := 0 TO Internal.col2-1 DO
		    FOR Internal.i1 := 0 TO Internal.row1-1 DO
				brsmemcpy(ADR(Internal.result),pB+(Internal.i1*Internal.col2+Internal.i3)*8,8);
		        FOR Internal.i2 := 0 TO Internal.i1-1 DO
					brsmemcpy(ADR(Internal.temp1),pL+(Internal.i1*Internal.col1+Internal.i2)*8,8);
					brsmemcpy(ADR(Internal.temp2),pOut+(Internal.i2*Internal.col2+Internal.i3)*8,8);
		            Internal.result := Internal.result - Internal.temp1*Internal.temp2;
		        END_FOR;
				brsmemcpy(ADR(Internal.temp1),pL+(Internal.i1*Internal.col1+Internal.i1)*8,8);
		        Internal.result 	:= Internal.result/Internal.temp1;
				brsmemcpy(pOut+(Internal.i1*Internal.col2+Internal.i3)*8,ADR(Internal.result),8);
		    END_FOR;
		    FOR Internal.i1 := Internal.row1-1 TO 0 BY -1 DO
				brsmemcpy(ADR(Internal.result),pOut+(Internal.i1*Internal.col2+Internal.i3)*8,8);
		        FOR Internal.i2 := Internal.i1+1 TO Internal.row1-1 DO
					brsmemcpy(ADR(Internal.temp1),pL+(Internal.i2*Internal.col1+Internal.i1)*8,8);
					brsmemcpy(ADR(Internal.temp2),pOut+(Internal.i2*Internal.col2+Internal.i3)*8,8);
		            Internal.result := Internal.result - Internal.temp1*Internal.temp2;
		        END_FOR;
				brsmemcpy(ADR(Internal.temp1),pL+(Internal.i1*Internal.col1+Internal.i1)*8,8);
		        Internal.result 	:= Internal.result/Internal.temp1;
				brsmemcpy(pOut+(Internal.i1*Internal.col2+Internal.i3)*8,ADR(Internal.result),8);
		    END_FOR;
		END_FOR;
	END_IF;
END_FUNCTION
```

#### HA_Matrix_RLS.st
```iecst
(* Recursive Least Squares Update *)
FUNCTION HA_Matrix_RLS
	HA_Matrix_RLS	 				:= TRUE;
	brsmemset(ADR(Internal),0,SIZEOF(Internal));
	Internal.sizeArray				:= SIZEOF(LREAL)*(MAX_HA_MATRIX_ARRAY_IDX+1);
	Internal.sizeTotal				:= Internal.sizeArray + SIZEOF(DINT)*2;
	brsmemcpy(ADR(Internal.row1),pTheta+Internal.sizeArray,4);
	brsmemcpy(ADR(Internal.col1),pTheta+Internal.sizeArray+4,4);
	brsmemcpy(ADR(Internal.row2),pP+Internal.sizeArray,4);
	brsmemcpy(ADR(Internal.col2),pP+Internal.sizeArray+4,4);
	brsmemcpy(ADR(Internal.row3),pX+Internal.sizeArray,4);
	brsmemcpy(ADR(Internal.col3),pX+Internal.sizeArray+4,4);
	IF pTheta = 0 OR pP = 0 OR pX = 0 OR Internal.row1 = 0 OR Internal.col1 = 0 OR Internal.row2 = 0 OR Internal.col2 = 0 OR Internal.row3 = 0 OR Internal.col3 = 0 OR Internal.col1 <> 1 OR Internal.row2 <> Internal.col2 OR Internal.row1 <> Internal.row2 OR Internal.row3 <> Internal.row1 OR Internal.col3 <> 1 OR Internal.row1*Internal.col1 > MAX_HA_MATRIX_ARRAY_IDX+1 OR Internal.row2*Internal.col2 > MAX_HA_MATRIX_ARRAY_IDX+1 OR Lambda <= 0.0 OR Lambda > 1.0 THEN
		HA_Matrix_RLS	 			:= FALSE;
	ELSE
		Internal.temp1 				:= 0.0;
		FOR Internal.i1 := 0 TO Internal.row1-1 DO
			Internal.temp2 			:= 0.0;
		    FOR Internal.i2 := 0 TO Internal.row2-1 DO
				brsmemcpy(ADR(Internal.temp3),pP+(Internal.i1*Internal.col2+Internal.i2)*8,8);
				brsmemcpy(ADR(Internal.temp4),pX+(Internal.i2*Internal.col3)*8,8);
		        Internal.temp2 		:= Internal.temp2 + Internal.temp3*Internal.temp4;
		    END_FOR;
			brsmemcpy(pTemp+(Internal.i1*1)*8,ADR(Internal.temp2),8);
			brsmemcpy(ADR(Internal.temp3),pX+(Internal.i1*Internal.col3)*8,8);
			Internal.temp1 			:= Internal.temp1 + Internal.temp3*Internal.temp2;
		END_FOR;
		Internal.temp1 				:= Lambda + Internal.temp1;
		IF ABS(Internal.temp1) < 1.0e-10 THEN
		    HA_Matrix_RLS	 		:= FALSE;
		    RETURN;
		END_IF;
		Internal.result 			:= 0.0;
		FOR Internal.i1 := 0 TO Internal.row1-1 DO
			brsmemcpy(ADR(Internal.temp2),pX+(Internal.i1*Internal.col3)*8,8);
			brsmemcpy(ADR(Internal.temp3),pTheta+(Internal.i1*Internal.col1)*8,8);
		    Internal.result 		:= Internal.result + Internal.temp2*Internal.temp3;
		END_FOR;
		Internal.result 			:= Y - Internal.result;
		FOR Internal.i1 := 0 TO Internal.row1-1 DO
			brsmemcpy(ADR(Internal.temp2),pTemp+(Internal.i1*1)*8,8);
		    Internal.temp3 			:= Internal.temp2/Internal.temp1;
			brsmemcpy(ADR(Internal.temp4),pTheta+(Internal.i1*Internal.col1)*8,8);
			Internal.temp4 			:= Internal.temp4 + Internal.temp3*Internal.result;
			brsmemcpy(pTheta+(Internal.i1*Internal.col1)*8,ADR(Internal.temp4),8);
		END_FOR;
		FOR Internal.i1 := 0 TO Internal.row2-1 DO
		    FOR Internal.i2 := 0 TO Internal.col2-1 DO
				Internal.temp2 		:= 0.0;
		        FOR Internal.i3 := 0 TO Internal.row2-1 DO
					brsmemcpy(ADR(Internal.temp3),pTemp+(Internal.i1*1)*8,8);
					brsmemcpy(ADR(Internal.temp4),pX+(Internal.i3*Internal.col3)*8,8);
					brsmemcpy(ADR(Internal.temp5),pP+(Internal.i3*Internal.col2+Internal.i2)*8,8);
		            Internal.temp2 	:= Internal.temp2 + Internal.temp3*Internal.temp4*Internal.temp5;
		        END_FOR;
				brsmemcpy(ADR(Internal.temp3),pP+(Internal.i1*Internal.col2+Internal.i2)*8,8);
		        Internal.result 	:= (Internal.temp3 - Internal.temp2/Internal.temp1)/Lambda;
				brsmemcpy(pP+(Internal.i1*Internal.col2+Internal.i2)*8,ADR(Internal.result),8);
		    END_FOR;
		END_FOR;
	END_IF;
END_FUNCTION
```

#### HA_Matrix_XtX.st
```iecst
(* Normal Equation X'X *)
FUNCTION HA_Matrix_XtX
	HA_Matrix_XtX	 				:= TRUE;
	brsmemset(ADR(Internal),0,SIZEOF(Internal));
	Internal.sizeArray				:= SIZEOF(LREAL)*(MAX_HA_MATRIX_ARRAY_IDX+1);
	Internal.sizeTotal				:= Internal.sizeArray + SIZEOF(DINT)*2;
	brsmemcpy(ADR(Internal.row1),pX+Internal.sizeArray,4);
	brsmemcpy(ADR(Internal.col1),pX+Internal.sizeArray+4,4);
	Internal.row2					:= Internal.col1;
	Internal.col2					:= Internal.col1;
	IF pX = 0 OR pOut = 0 OR Internal.row1 = 0 OR Internal.col1 = 0 OR Internal.row1*Internal.col1 > MAX_HA_MATRIX_ARRAY_IDX+1 OR Internal.row2*Internal.col2 > MAX_HA_MATRIX_ARRAY_IDX+1 THEN
		HA_Matrix_XtX	 			:= FALSE;
	ELSE
		brsmemset(pOut,0,Internal.sizeTotal);
		brsmemcpy(pOut+Internal.sizeArray,ADR(Internal.row2),4);
		brsmemcpy(pOut+Internal.sizeArray+4,ADR(Internal.col2),4);
		FOR Internal.i1 := 0 TO Internal.col1-1 DO
		    FOR Internal.i2 := 0 TO Internal.col1-1 DO
		        Internal.result 	:= 0.0;
		        FOR Internal.i3 := 0 TO Internal.row1-1 DO
					brsmemcpy(ADR(Internal.temp1),pX+(Internal.i3*Internal.col1+Internal.i1)*8,8);
					brsmemcpy(ADR(Internal.temp2),pX+(Internal.i3*Internal.col1+Internal.i2)*8,8);
		            Internal.result := Internal.result + Internal.temp1*Internal.temp2;
		        END_FOR;
				brsmemcpy(pOut+(Internal.i1*Internal.col2+Internal.i2)*8,ADR(Internal.result),8);
		    END_FOR;
		END_FOR;
	END_IF;
END_FUNCTION
```

#### HA_Matrix_XtY.st
```iecst
(* Normal Equation X'Y *)
FUNCTION HA_Matrix_XtY
	HA_Matrix_XtY	 				:= TRUE;
	brsmemset(ADR(Internal),0,SIZEOF(Internal));
	Internal.sizeArray				:= SIZEOF(LREAL)*(MAX_HA_MATRIX_ARRAY_IDX+1);
	Internal.sizeTotal				:= Internal.sizeArray + SIZEOF(DINT)*2;
	brsmemcpy(ADR(Internal.row1),pX+Internal.sizeArray,4);
	brsmemcpy(ADR(Internal.col1),pX+Internal.sizeArray+4,4);
	brsmemcpy(ADR(Internal.row2),pY+Internal.sizeArray,4);
	brsmemcpy(ADR(Internal.col2),pY+Internal.sizeArray+4,4);
	Internal.row3					:= Internal.col1;
	Internal.col3					:= Internal.col2;
	IF pX = 0 OR pY = 0 OR pOut = 0 OR Internal.row1 = 0 OR Internal.col1 = 0 OR Internal.row2 = 0 OR Internal.col2 = 0 OR Internal.row1 <> Internal.row2 OR Internal.row1*Internal.col1 > MAX_HA_MATRIX_ARRAY_IDX+1 OR Internal.row2*Internal.col2 > MAX_HA_MATRIX_ARRAY_IDX+1 OR Internal.row3*Internal.col3 > MAX_HA_MATRIX_ARRAY_IDX+1 THEN
		HA_Matrix_XtY	 			:= FALSE;
	ELSE
		brsmemset(pOut,0,Internal.sizeTotal);
		brsmemcpy(pOut+Internal.sizeArray,ADR(Internal.row3),4);
		brsmemcpy(pOut+Internal.sizeArray+4,ADR(Internal.col3),4);
		FOR Internal.i1 := 0 TO Internal.col1-1 DO
		    FOR Internal.i2 := 0 TO Internal.col2-1 DO
		        Internal.result 	:= 0.0;
		        FOR Internal.i3 := 0 TO Internal.row1-1 DO
					brsmemcpy(ADR(Internal.temp1),pX+(Internal.i3*Internal.col1+Internal.i1)*8,8);
					brsmemcpy(ADR(Internal.temp2),pY+(Internal.i3*Internal.col2+Internal.i2)*8,8);
		            Internal.result := Internal.result + Internal.temp1*Internal.temp2;
		        END_FOR;
				brsmemcpy(pOut+(Internal.i1*Internal.col3+Internal.i2)*8,ADR(Internal.result),8);
		    END_FOR;
		END_FOR;
	END_IF;
END_FUNCTION
```

#### HA_Matrix_AddRidge.st
```iecst
(* Add Ridge Penalty *)
FUNCTION HA_Matrix_AddRidge
	HA_Matrix_AddRidge	 			:= TRUE;
	brsmemset(ADR(Internal),0,SIZEOF(Internal));
	Internal.sizeArray				:= SIZEOF(LREAL)*(MAX_HA_MATRIX_ARRAY_IDX+1);
	Internal.sizeTotal				:= Internal.sizeArray + SIZEOF(DINT)*2;
	brsmemcpy(ADR(Internal.row1),pInOut+Internal.sizeArray,4);
	brsmemcpy(ADR(Internal.col1),pInOut+Internal.sizeArray+4,4);
	IF pInOut = 0 OR Internal.row1 = 0 OR Internal.col1 = 0 OR Internal.row1 <> Internal.col1 OR Internal.row1*Internal.col1 > MAX_HA_MATRIX_ARRAY_IDX+1 OR Lambda < 0.0 THEN
		HA_Matrix_AddRidge	 		:= FALSE;
	ELSE
		FOR Internal.i1 := 0 TO Internal.row1-1 DO
			brsmemcpy(ADR(Internal.temp1),pInOut+(Internal.i1*Internal.col1+Internal.i1)*8,8);
		    Internal.temp1 			:= Internal.temp1 + Lambda;
			brsmemcpy(pInOut+(Internal.i1*Internal.col1+Internal.i1)*8,ADR(Internal.temp1),8);
		END_FOR;
	END_IF;
END_FUNCTION
```

#### HA_Matrix_RLS_Init.st
```iecst
(* Initialize RLS *)
FUNCTION HA_Matrix_RLS_Init
	HA_Matrix_RLS_Init	 			:= TRUE;
	brsmemset(ADR(Internal),0,SIZEOF(Internal));
	Internal.sizeArray				:= SIZEOF(LREAL)*(MAX_HA_MATRIX_ARRAY_IDX+1);
	Internal.sizeTotal				:= Internal.sizeArray + SIZEOF(DINT)*2;
	brsmemcpy(ADR(Internal.row1),pTheta+Internal.sizeArray,4);
	brsmemcpy(ADR(Internal.col1),pTheta+Internal.sizeArray+4,4);
	brsmemcpy(ADR(Internal.row2),pP+Internal.sizeArray,4);
	brsmemcpy(ADR(Internal.col2),pP+Internal.sizeArray+4,4);
	IF pTheta = 0 OR pP = 0 OR Internal.row1 = 0 OR Internal.col1 = 0 OR Internal.row2 = 0 OR Internal.col2 = 0 OR Internal.col1 <> 1 OR Internal.row2 <> Internal.col2 OR Internal.row1 <> Internal.row2 OR Internal.row1*Internal.col1 > MAX_HA_MATRIX_ARRAY_IDX+1 OR Internal.row2*Internal.col2 > MAX_HA_MATRIX_ARRAY_IDX+1 OR InitVariance <= 0.0 THEN
		HA_Matrix_RLS_Init	 		:= FALSE;
	ELSE
		FOR Internal.i1 := 0 TO Internal.row1-1 DO
			Internal.temp1 			:= 0.0;
			brsmemcpy(pTheta+(Internal.i1*Internal.col1)*8,ADR(Internal.temp1),8);
		END_FOR;
		FOR Internal.i1 := 0 TO Internal.row2-1 DO
		    FOR Internal.i2 := 0 TO Internal.col2-1 DO
				Internal.temp1 		:= 0.0;
				IF Internal.i1 = Internal.i2 THEN
					Internal.temp1 	:= InitVariance;
				END_IF;
				brsmemcpy(pP+(Internal.i1*Internal.col2+Internal.i2)*8,ADR(Internal.temp1),8);
		    END_FOR;
		END_FOR;
	END_IF;
END_FUNCTION
```

#### HA_Matrix_BuildLags.st
```iecst
(* Build Lag Matrix *)
FUNCTION HA_Matrix_BuildLags
	HA_Matrix_BuildLags	 			:= TRUE;
	brsmemset(ADR(Internal),0,SIZEOF(Internal));
	Internal.sizeArray				:= SIZEOF(LREAL)*(MAX_HA_MATRIX_ARRAY_IDX+1);
	Internal.sizeTotal				:= Internal.sizeArray + SIZEOF(DINT)*2;
	brsmemcpy(ADR(Internal.row1),pY_history+Internal.sizeArray,4);
	brsmemcpy(ADR(Internal.col1),pY_history+Internal.sizeArray+4,4);
	IF pU_history <> 0 THEN
		brsmemcpy(ADR(Internal.row2),pU_history+Internal.sizeArray,4);
		brsmemcpy(ADR(Internal.col2),pU_history+Internal.sizeArray+4,4);
	ELSE
		Internal.row2 				:= 0;
		Internal.col2 				:= 0;
	END_IF;
	Internal.row3					:= NumOutputs*LagOrder + NumInputs*LagOrder;
	Internal.col3					:= 1;
	IF pY_history = 0 OR pOut = 0 OR LagOrder = 0 OR NumOutputs = 0 OR Internal.row1 = 0 OR Internal.col1 = 0 OR Internal.row1 < NumOutputs*LagOrder OR Internal.col1 <> 1 OR Internal.row3*Internal.col3 > MAX_HA_MATRIX_ARRAY_IDX+1 THEN
		HA_Matrix_BuildLags	 		:= FALSE;
	ELSE
		IF pU_history <> 0 THEN
			IF NumInputs = 0 OR Internal.row2 = 0 OR Internal.col2 = 0 OR Internal.row2 < NumInputs*LagOrder OR Internal.col2 <> 1 THEN
				HA_Matrix_BuildLags	 := FALSE;
				RETURN;
			END_IF;
		END_IF;
		brsmemset(pOut,0,Internal.sizeTotal);
		brsmemcpy(pOut+Internal.sizeArray,ADR(Internal.row3),4);
		brsmemcpy(pOut+Internal.sizeArray+4,ADR(Internal.col3),4);
		Internal.i4 				:= 0;
		FOR Internal.i1 := 0 TO LagOrder-1 DO
		    FOR Internal.i2 := 0 TO NumOutputs-1 DO
				brsmemcpy(ADR(Internal.temp1),pY_history+(Internal.i1*NumOutputs+Internal.i2)*8,8);
				brsmemcpy(pOut+Internal.i4*8,ADR(Internal.temp1),8);
				Internal.i4 			:= Internal.i4 + 1;
		    END_FOR;
		END_FOR;
		IF pU_history <> 0 AND NumInputs > 0 THEN
			FOR Internal.i1 := 0 TO LagOrder-1 DO
			    FOR Internal.i2 := 0 TO NumInputs-1 DO
					brsmemcpy(ADR(Internal.temp1),pU_history+(Internal.i1*NumInputs+Internal.i2)*8,8);
					brsmemcpy(pOut+Internal.i4*8,ADR(Internal.temp1),8);
					Internal.i4 		:= Internal.i4 + 1;
			    END_FOR;
			END_FOR;
		END_IF;
	END_IF;
END_FUNCTION
```

#### HA_Matrix_RollingUpdate.st
```iecst
(* Rolling Buffer Update *)
FUNCTION HA_Matrix_RollingUpdate
	HA_Matrix_RollingUpdate	 		:= TRUE;
	brsmemset(ADR(Internal),0,SIZEOF(Internal));
	Internal.sizeArray				:= SIZEOF(LREAL)*(MAX_HA_MATRIX_ARRAY_IDX+1);
	Internal.sizeTotal				:= Internal.sizeArray + SIZEOF(DINT)*2;
	brsmemcpy(ADR(Internal.row1),pBuffer+Internal.sizeArray,4);
	brsmemcpy(ADR(Internal.col1),pBuffer+Internal.sizeArray+4,4);
	IF pBuffer = 0 OR Internal.row1 = 0 OR Internal.col1 = 0 OR Internal.row1*Internal.col1 > MAX_HA_MATRIX_ARRAY_IDX+1 THEN
		HA_Matrix_RollingUpdate	 	:= FALSE;
	ELSE
		FOR Internal.i1 := Internal.row1*Internal.col1-1 TO 1 BY -1 DO
			brsmemcpy(ADR(Internal.temp1),pBuffer+(Internal.i1-1)*8,8);
			brsmemcpy(pBuffer+Internal.i1*8,ADR(Internal.temp1),8);
		END_FOR;
		brsmemcpy(pBuffer,ADR(NewValue),8);
	END_IF;
END_FUNCTION
```

#### HA_Matrix_Predict.st
```iecst
(* Predict *)
FUNCTION HA_Matrix_Predict
	HA_Matrix_Predict	 			:= TRUE;
	brsmemset(ADR(Internal),0,SIZEOF(Internal));
	Internal.sizeArray				:= SIZEOF(LREAL)*(MAX_HA_MATRIX_ARRAY_IDX+1);
	Internal.sizeTotal				:= Internal.sizeArray + SIZEOF(DINT)*2;
	brsmemcpy(ADR(Internal.row1),pX+Internal.sizeArray,4);
	brsmemcpy(ADR(Internal.col1),pX+Internal.sizeArray+4,4);
	brsmemcpy(ADR(Internal.row2),pBeta+Internal.sizeArray,4);
	brsmemcpy(ADR(Internal.col2),pBeta+Internal.sizeArray+4,4);
	Internal.row3					:= Internal.row1;
	Internal.col3					:= Internal.col2;
	IF pX = 0 OR pBeta = 0 OR pOut = 0 OR Internal.row1 = 0 OR Internal.col1 = 0 OR Internal.row2 = 0 OR Internal.col2 = 0 OR Internal.col1 <> Internal.row2 OR Internal.row1*Internal.col1 > MAX_HA_MATRIX_ARRAY_IDX+1 OR Internal.row2*Internal.col2 > MAX_HA_MATRIX_ARRAY_IDX+1 OR Internal.row3*Internal.col3 > MAX_HA_MATRIX_ARRAY_IDX+1 THEN
		HA_Matrix_Predict	 		:= FALSE;
	ELSE
		brsmemset(pOut,0,Internal.sizeTotal);
		brsmemcpy(pOut+Internal.sizeArray,ADR(Internal.row3),4);
		brsmemcpy(pOut+Internal.sizeArray+4,ADR(Internal.col3),4);
		FOR Internal.i1 := 0 TO Internal.row1-1 DO
		    FOR Internal.i2 := 0 TO Internal.col2-1 DO
		        Internal.result 	:= 0.0;
		        FOR Internal.i3 := 0 TO Internal.col1-1 DO
					brsmemcpy(ADR(Internal.temp1),pX+(Internal.i1*Internal.col1+Internal.i3)*8,8);
					brsmemcpy(ADR(Internal.temp2),pBeta+(Internal.i3*Internal.col2+Internal.i2)*8,8);
		            Internal.result := Internal.result + Internal.temp1*Internal.temp2;
		        END_FOR;
				brsmemcpy(pOut+(Internal.i1*Internal.col3+Internal.i2)*8,ADR(Internal.result),8);
		    END_FOR;
		END_FOR;
	END_IF;
END_FUNCTION
```

#### HA_Matrix_RMSE.st
```iecst
(* Root Mean Square Error *)
FUNCTION HA_Matrix_RMSE
	HA_Matrix_RMSE	 				:= 0.0;
	brsmemset(ADR(Internal),0,SIZEOF(Internal));
	Internal.sizeArray				:= SIZEOF(LREAL)*(MAX_HA_MATRIX_ARRAY_IDX+1);
	Internal.sizeTotal				:= Internal.sizeArray + SIZEOF(DINT)*2;
	brsmemcpy(ADR(Internal.row1),pY_true+Internal.sizeArray,4);
	brsmemcpy(ADR(Internal.col1),pY_true+Internal.sizeArray+4,4);
	brsmemcpy(ADR(Internal.row2),pY_pred+Internal.sizeArray,4);
	brsmemcpy(ADR(Internal.col2),pY_pred+Internal.sizeArray+4,4);
	IF pY_true = 0 OR pY_pred = 0 OR Internal.row1 = 0 OR Internal.col1 = 0 OR Internal.row2 = 0 OR Internal.col2 = 0 OR Internal.row1 <> Internal.row2 OR Internal.col1 <> Internal.col2 OR Internal.row1*Internal.col1 > MAX_HA_MATRIX_ARRAY_IDX+1 THEN
		HA_Matrix_RMSE	 			:= 0.0;
	ELSE
		Internal.result 			:= 0.0;
		FOR Internal.i1 := 0 TO Internal.row1-1 DO
		    FOR Internal.i2 := 0 TO Internal.col1-1 DO
				brsmemcpy(ADR(Internal.temp1),pY_true+(Internal.i1*Internal.col1+Internal.i2)*8,8);
				brsmemcpy(ADR(Internal.temp2),pY_pred+(Internal.i1*Internal.col1+Internal.i2)*8,8);
		        Internal.temp3 		:= Internal.temp1 - Internal.temp2;
		        Internal.result 	:= Internal.result + Internal.temp3*Internal.temp3;
		    END_FOR;
		END_FOR;
		Internal.result 			:= Internal.result/DINT_TO_LREAL(Internal.row1*Internal.col1);
		HA_Matrix_RMSE	 			:= SQRT(Internal.result);
	END_IF;
END_FUNCTION
```

#### HA_Matrix_Residuals.st
```iecst
(* Residuals *)
FUNCTION HA_Matrix_Residuals
	HA_Matrix_Residuals	 			:= TRUE;
	brsmemset(ADR(Internal),0,SIZEOF(Internal));
	Internal.sizeArray				:= SIZEOF(LREAL)*(MAX_HA_MATRIX_ARRAY_IDX+1);
	Internal.sizeTotal				:= Internal.sizeArray + SIZEOF(DINT)*2;
	brsmemcpy(ADR(Internal.row1),pY_true+Internal.sizeArray,4);
	brsmemcpy(ADR(Internal.col1),pY_true+Internal.sizeArray+4,4);
	brsmemcpy(ADR(Internal.row2),pY_pred+Internal.sizeArray,4);
	brsmemcpy(ADR(Internal.col2),pY_pred+Internal.sizeArray+4,4);
	IF pY_true = 0 OR pY_pred = 0 OR pOut = 0 OR Internal.row1 = 0 OR Internal.col1 = 0 OR Internal.row2 = 0 OR Internal.col2 = 0 OR Internal.row1*Internal.col1 > MAX_HA_MATRIX_ARRAY_IDX+1 OR Internal.row2*Internal.col2 > MAX_HA_MATRIX_ARRAY_IDX+1 OR Internal.row1 <> Internal.row2 OR Internal.col1 <> Internal.col2 THEN
		HA_Matrix_Residuals	 		:= FALSE;
	ELSE
		brsmemset(pOut,0,Internal.sizeTotal);
		brsmemcpy(pOut+Internal.sizeArray,ADR(Internal.row1),4);
		brsmemcpy(pOut+Internal.sizeArray+4,ADR(Internal.col1),4);
		FOR Internal.i1 := 0 TO Internal.row1-1 DO
		    FOR Internal.i2 := 0 TO Internal.col1-1 DO
				brsmemcpy(ADR(Internal.temp1),pY_true+(Internal.i1*Internal.col1+Internal.i2)*8,8);
				brsmemcpy(ADR(Internal.temp2),pY_pred+(Internal.i1*Internal.col1+Internal.i2)*8,8);
		        Internal.result 	:= Internal.temp1 - Internal.temp2;
				brsmemcpy(pOut+(Internal.i1*Internal.col1+Internal.i2)*8,ADR(Internal.result),8);
		    END_FOR;
		END_FOR;
	END_IF;
END_FUNCTION
```

#### HA_Matrix_R2Score.st
```iecst
(* R-squared Score *)
FUNCTION HA_Matrix_R2Score
	HA_Matrix_R2Score	 			:= 0.0;
	brsmemset(ADR(Internal),0,SIZEOF(Internal));
	Internal.sizeArray				:= SIZEOF(LREAL)*(MAX_HA_MATRIX_ARRAY_IDX+1);
	Internal.sizeTotal				:= Internal.sizeArray + SIZEOF(DINT)*2;
	brsmemcpy(ADR(Internal.row1),pY_true+Internal.sizeArray,4);
	brsmemcpy(ADR(Internal.col1),pY_true+Internal.sizeArray+4,4);
	brsmemcpy(ADR(Internal.row2),pY_pred+Internal.sizeArray,4);
	brsmemcpy(ADR(Internal.col2),pY_pred+Internal.sizeArray+4,4);
	IF pY_true = 0 OR pY_pred = 0 OR Internal.row1 = 0 OR Internal.col1 = 0 OR Internal.row2 = 0 OR Internal.col2 = 0 OR Internal.row1 <> Internal.row2 OR Internal.col1 <> Internal.col2 OR Internal.row1*Internal.col1 > MAX_HA_MATRIX_ARRAY_IDX+1 THEN
		HA_Matrix_R2Score	 		:= 0.0;
	ELSE
		Internal.temp1 				:= 0.0;
		FOR Internal.i1 := 0 TO Internal.row1-1 DO
		    FOR Internal.i2 := 0 TO Internal.col1-1 DO
				brsmemcpy(ADR(Internal.temp2),pY_true+(Internal.i1*Internal.col1+Internal.i2)*8,8);
		        Internal.temp1 		:= Internal.temp1 + Internal.temp2;
		    END_FOR;
		END_FOR;
		Internal.temp1 				:= Internal.temp1/DINT_TO_LREAL(Internal.row1*Internal.col1);
		Internal.temp2 				:= 0.0;
		Internal.temp3 				:= 0.0;
		FOR Internal.i1 := 0 TO Internal.row1-1 DO
		    FOR Internal.i2 := 0 TO Internal.col1-1 DO
				brsmemcpy(ADR(Internal.temp4),pY_true+(Internal.i1*Internal.col1+Internal.i2)*8,8);
				brsmemcpy(ADR(Internal.temp5),pY_pred+(Internal.i1*Internal.col1+Internal.i2)*8,8);
		        Internal.result 	:= Internal.temp4 - Internal.temp5;
		        Internal.temp2 		:= Internal.temp2 + Internal.result*Internal.result;
		        Internal.result 	:= Internal.temp4 - Internal.temp1;
		        Internal.temp3 		:= Internal.temp3 + Internal.result*Internal.result;
		    END_FOR;
		END_FOR;
		IF ABS(Internal.temp3) < 1.0e-10 THEN
			HA_Matrix_R2Score	 	:= 0.0;
		ELSE
			HA_Matrix_R2Score	 	:= 1.0 - Internal.temp2/Internal.temp3;
		END_IF;
	END_IF;
END_FUNCTION
```

#### HA_Matrix_Standardize.st
```iecst
(* Standardize Features *)
FUNCTION HA_Matrix_Standardize
	HA_Matrix_Standardize	 		:= TRUE;
	brsmemset(ADR(Internal),0,SIZEOF(Internal));
	Internal.sizeArray				:= SIZEOF(LREAL)*(MAX_HA_MATRIX_ARRAY_IDX+1);
	Internal.sizeTotal				:= Internal.sizeArray + SIZEOF(DINT)*2;
	brsmemcpy(ADR(Internal.row1),pX+Internal.sizeArray,4);
	brsmemcpy(ADR(Internal.col1),pX+Internal.sizeArray+4,4);
	brsmemcpy(ADR(Internal.row2),pMean+Internal.sizeArray,4);
	brsmemcpy(ADR(Internal.col2),pMean+Internal.sizeArray+4,4);
	brsmemcpy(ADR(Internal.row3),pStd+Internal.sizeArray,4);
	brsmemcpy(ADR(Internal.col3),pStd+Internal.sizeArray+4,4);
	IF pX = 0 OR pMean = 0 OR pStd = 0 OR Internal.row1 = 0 OR Internal.col1 = 0 OR Internal.row2 = 0 OR Internal.col2 = 0 OR Internal.row3 = 0 OR Internal.col3 = 0 OR Internal.row1*Internal.col1 > MAX_HA_MATRIX_ARRAY_IDX+1 OR Internal.row2 <> Internal.col1 OR Internal.col2 <> 1 OR Internal.row3 <> Internal.col1 OR Internal.col3 <> 1 THEN
		HA_Matrix_Standardize	 	:= FALSE;
	ELSE
		IF Mode = 0 THEN
			FOR Internal.i2 := 0 TO Internal.col1-1 DO
				Internal.temp1 		:= 0.0;
				FOR Internal.i1 := 0 TO Internal.row1-1 DO
					brsmemcpy(ADR(Internal.temp2),pX+(Internal.i1*Internal.col1+Internal.i2)*8,8);
					Internal.temp1 	:= Internal.temp1 + Internal.temp2;
				END_FOR;
				Internal.temp1 		:= Internal.temp1/DINT_TO_LREAL(Internal.row1);
				brsmemcpy(pMean+Internal.i2*8,ADR(Internal.temp1),8);
			END_FOR;
			FOR Internal.i2 := 0 TO Internal.col1-1 DO
				brsmemcpy(ADR(Internal.temp1),pMean+Internal.i2*8,8);
				Internal.temp2 		:= 0.0;
				FOR Internal.i1 := 0 TO Internal.row1-1 DO
					brsmemcpy(ADR(Internal.temp3),pX+(Internal.i1*Internal.col1+Internal.i2)*8,8);
					Internal.temp4 	:= Internal.temp3 - Internal.temp1;
					Internal.temp2 	:= Internal.temp2 + Internal.temp4*Internal.temp4;
				END_FOR;
				Internal.temp2 		:= Internal.temp2/DINT_TO_LREAL(Internal.row1);
				Internal.temp2 		:= SQRT(Internal.temp2);
				IF Internal.temp2 < 1.0e-10 THEN
					Internal.temp2 	:= 1.0;
				END_IF;
				brsmemcpy(pStd+Internal.i2*8,ADR(Internal.temp2),8);
			END_FOR;
		END_IF;
		FOR Internal.i1 := 0 TO Internal.row1-1 DO
		    FOR Internal.i2 := 0 TO Internal.col1-1 DO
				brsmemcpy(ADR(Internal.temp1),pX+(Internal.i1*Internal.col1+Internal.i2)*8,8);
				brsmemcpy(ADR(Internal.temp2),pMean+Internal.i2*8,8);
				brsmemcpy(ADR(Internal.temp3),pStd+Internal.i2*8,8);
		        Internal.result 	:= (Internal.temp1 - Internal.temp2)/Internal.temp3;
				brsmemcpy(pX+(Internal.i1*Internal.col1+Internal.i2)*8,ADR(Internal.result),8);
		    END_FOR;
		END_FOR;
	END_IF;
END_FUNCTION
```

#### HA_Matrix_PolyExpand.st
```iecst
(* Polynomial Feature Expansion *)
FUNCTION HA_Matrix_PolyExpand
	HA_Matrix_PolyExpand	 		:= TRUE;
	brsmemset(ADR(Internal),0,SIZEOF(Internal));
	Internal.sizeArray				:= SIZEOF(LREAL)*(MAX_HA_MATRIX_ARRAY_IDX+1);
	Internal.sizeTotal				:= Internal.sizeArray + SIZEOF(UDINT)*2;
	brsmemcpy(ADR(Internal.row1),pX+Internal.sizeArray,4);
	brsmemcpy(ADR(Internal.col1),pX+Internal.sizeArray+4,4);
	IF Order = 2 THEN
		Internal.col2 			:= Internal.col1 + (Internal.col1*(Internal.col1+1))/2;
	ELSIF Order = 3 THEN
		Internal.col2 			:= Internal.col1 + (Internal.col1*(Internal.col1+1))/2 + (Internal.col1*(Internal.col1+1)*(Internal.col1+2))/6;
	ELSE
		Internal.col2 			:= Internal.col1;
	END_IF;
	Internal.row2					:= Internal.row1;
	IF pX = 0 OR pOut = 0 OR Internal.row1 = 0 OR Internal.col1 = 0 OR Order < 1 OR Order > 3 OR Internal.row1*Internal.col1 > MAX_HA_MATRIX_ARRAY_IDX+1 OR Internal.row2*Internal.col2 > MAX_HA_MATRIX_ARRAY_IDX+1 THEN
		HA_Matrix_PolyExpand	 	:= FALSE;
	ELSE
		brsmemset(pOut,0,Internal.sizeTotal);
		brsmemcpy(pOut+Internal.sizeArray,ADR(Internal.row2),4);
		brsmemcpy(pOut+Internal.sizeArray+4,ADR(Internal.col2),4);
		FOR Internal.i1 := 0 TO Internal.row1-1 DO
			Internal.i4 			:= 0;
		    FOR Internal.i2 := 0 TO Internal.col1-1 DO
				brsmemcpy(ADR(Internal.temp1),pX+(Internal.i1*Internal.col1+Internal.i2)*8,8);
				brsmemcpy(pOut+(Internal.i1*Internal.col2+Internal.i4)*8,ADR(Internal.temp1),8);
				Internal.i4 		:= Internal.i4 + 1;
		    END_FOR;
			IF Order >= 2 THEN
				FOR Internal.i2 := 0 TO Internal.col1-1 DO
				    FOR Internal.i3 := Internal.i2 TO Internal.col1-1 DO
						brsmemcpy(ADR(Internal.temp1),pX+(Internal.i1*Internal.col1+Internal.i2)*8,8);
						brsmemcpy(ADR(Internal.temp2),pX+(Internal.i1*Internal.col1+Internal.i3)*8,8);
						Internal.result := Internal.temp1*Internal.temp2;
						brsmemcpy(pOut+(Internal.i1*Internal.col2+Internal.i4)*8,ADR(Internal.result),8);
						Internal.i4 	:= Internal.i4 + 1;
				    END_FOR;
				END_FOR;
			END_IF;
			IF Order >= 3 THEN
				FOR Internal.i2 := 0 TO Internal.col1-1 DO
				    FOR Internal.i3 := Internal.i2 TO Internal.col1-1 DO
						FOR Internal.row3 := Internal.i3 TO Internal.col1-1 DO
							brsmemcpy(ADR(Internal.temp1),pX+(Internal.i1*Internal.col1+Internal.i2)*8,8);
							brsmemcpy(ADR(Internal.temp2),pX+(Internal.i1*Internal.col1+Internal.i3)*8,8);
							brsmemcpy(ADR(Internal.temp3),pX+(Internal.i1*Internal.col1+Internal.row3)*8,8);
							Internal.result := Internal.temp1*Internal.temp2*Internal.temp3;
							brsmemcpy(pOut+(Internal.i1*Internal.col2+Internal.i4)*8,ADR(Internal.result),8);
							Internal.i4 := Internal.i4 + 1;
						END_FOR;
				    END_FOR;
				END_FOR;
			END_IF;
		END_FOR;
	END_IF;
END_FUNCTION
```

#### HA_Matrix_Diff.st
```iecst
(* Calculate Differences *)
FUNCTION HA_Matrix_Diff
	HA_Matrix_Diff	 				:= TRUE;
	brsmemset(ADR(Internal),0,SIZEOF(Internal));
	Internal.sizeArray				:= SIZEOF(LREAL)*(MAX_HA_MATRIX_ARRAY_IDX+1);
	Internal.sizeTotal				:= Internal.sizeArray + SIZEOF(UDINT)*2;
	brsmemcpy(ADR(Internal.row1),pX+Internal.sizeArray,4);
	brsmemcpy(ADR(Internal.col1),pX+Internal.sizeArray+4,4);
	Internal.row2					:= Internal.row1 - 1;
	Internal.col2					:= Internal.col1;
	IF pX = 0 OR pOut = 0 OR Internal.row1 = 0 OR Internal.col1 = 0 OR Internal.row1 < 2 OR Internal.row1*Internal.col1 > MAX_HA_MATRIX_ARRAY_IDX+1 OR Internal.row2*Internal.col2 > MAX_HA_MATRIX_ARRAY_IDX+1 THEN
		HA_Matrix_Diff	 			:= FALSE;
	ELSE
		brsmemset(pOut,0,Internal.sizeTotal);
		brsmemcpy(pOut+Internal.sizeArray,ADR(Internal.row2),4);
		brsmemcpy(pOut+Internal.sizeArray+4,ADR(Internal.col2),4);
		FOR Internal.i1 := 0 TO Internal.row2-1 DO
		    FOR Internal.i2 := 0 TO Internal.col1-1 DO
				brsmemcpy(ADR(Internal.temp1),pX+((Internal.i1+1)*Internal.col1+Internal.i2)*8,8);
				brsmemcpy(ADR(Internal.temp2),pX+(Internal.i1*Internal.col1+Internal.i2)*8,8);
		        Internal.result 	:= Internal.temp1 - Internal.temp2;
				brsmemcpy(pOut+(Internal.i1*Internal.col2+Internal.i2)*8,ADR(Internal.result),8);
		    END_FOR;
		END_FOR;
	END_IF;
END_FUNCTION
```

#### HA_Matrix_AddBias.st
```iecst
(* Add Bias Column *)
FUNCTION HA_Matrix_AddBias
	HA_Matrix_AddBias	 			:= TRUE;
	brsmemset(ADR(Internal),0,SIZEOF(Internal));
	Internal.sizeArray				:= SIZEOF(LREAL)*(MAX_HA_MATRIX_ARRAY_IDX+1);
	Internal.sizeTotal				:= Internal.sizeArray + SIZEOF(UDINT)*2;
	brsmemcpy(ADR(Internal.row1),pX+Internal.sizeArray,4);
	brsmemcpy(ADR(Internal.col1),pX+Internal.sizeArray+4,4);
	Internal.row2					:= Internal.row1;
	Internal.col2					:= Internal.col1 + 1;
	IF pX = 0 OR pOut = 0 OR Internal.row1 = 0 OR Internal.col1 = 0 OR Internal.row1*Internal.col1 > MAX_HA_MATRIX_ARRAY_IDX+1 OR Internal.row2*Internal.col2 > MAX_HA_MATRIX_ARRAY_IDX+1 THEN
		HA_Matrix_AddBias	 		:= FALSE;
	ELSE
		brsmemset(pOut,0,Internal.sizeTotal);
		brsmemcpy(pOut+Internal.sizeArray,ADR(Internal.row2),4);
		brsmemcpy(pOut+Internal.sizeArray+4,ADR(Internal.col2),4);
		Internal.temp1 				:= 1.0;
		FOR Internal.i1 := 0 TO Internal.row1-1 DO
			brsmemcpy(pOut+(Internal.i1*Internal.col2)*8,ADR(Internal.temp1),8);
		    FOR Internal.i2 := 0 TO Internal.col1-1 DO
				brsmemcpy(ADR(Internal.temp2),pX+(Internal.i1*Internal.col1+Internal.i2)*8,8);
				brsmemcpy(pOut+(Internal.i1*Internal.col2+Internal.i2+1)*8,ADR(Internal.temp2),8);
		    END_FOR;
		END_FOR;
	END_IF;
END_FUNCTION
```

#### HA_Matrix_PredictMultiStep.st
```iecst
(* Multi-Step Prediction with Integration *)
FUNCTION HA_Matrix_PredictMultiStep
	HA_Matrix_PredictMultiStep	 	:= TRUE;
	brsmemset(ADR(Internal),0,SIZEOF(Internal));
	Internal.sizeArray				:= SIZEOF(LREAL)*(MAX_HA_MATRIX_ARRAY_IDX+1);
	Internal.sizeTotal				:= Internal.sizeArray + SIZEOF(UDINT)*2;
	brsmemcpy(ADR(Internal.row1),pState+Internal.sizeArray,4);
	brsmemcpy(ADR(Internal.col1),pState+Internal.sizeArray+4,4);
	brsmemcpy(ADR(Internal.row2),pBeta+Internal.sizeArray,4);
	brsmemcpy(ADR(Internal.col2),pBeta+Internal.sizeArray+4,4);
	brsmemcpy(ADR(Internal.row3),pHistory+Internal.sizeArray,4);
	brsmemcpy(ADR(Internal.col3),pHistory+Internal.sizeArray+4,4);
	Internal.row4					:= Steps;
	Internal.col4					:= Internal.col1;
	IF pState = 0 OR pBeta = 0 OR pHistory = 0 OR pOut = 0 OR pLagTemp = 0 OR Internal.row1 = 0 OR Internal.col1 = 0 OR Internal.row2 = 0 OR Internal.col2 = 0 OR Internal.row3 = 0 OR Internal.col3 = 0 OR Steps <= 0 OR LagOrder < 0 OR PolyOrder < 1 OR PolyOrder > 3 OR Internal.row1 <> 1 OR Internal.col3 <> 1 OR Internal.col2 <> Internal.col1 OR Internal.row4*Internal.col4 > MAX_HA_MATRIX_ARRAY_IDX+1 THEN
		HA_Matrix_PredictMultiStep	:= FALSE;
	ELSE
		brsmemset(pOut,0,Internal.sizeTotal);
		brsmemcpy(pOut+Internal.sizeArray,ADR(Internal.row4),4);
		brsmemcpy(pOut+Internal.sizeArray+4,ADR(Internal.col4),4);
		FOR Internal.i1 := 0 TO Internal.col1-1 DO
			brsmemcpy(ADR(Internal.temp1),pState+Internal.i1*8,8);
			brsmemcpy(pWorkState+Internal.i1*8,ADR(Internal.temp1),8);
		END_FOR;
		FOR Internal.i1 := 0 TO Internal.row3-1 DO
			brsmemcpy(ADR(Internal.temp1),pHistory+Internal.i1*8,8);
			brsmemcpy(pWorkHist+Internal.i1*8,ADR(Internal.temp1),8);
		END_FOR;
		FOR Internal.i1 := 0 TO Steps-1 DO
			Success := HA_Matrix_BuildLags(pWorkHist,0,LagOrder,Internal.col1,0,pLagTemp);
			IF NOT Success THEN
				HA_Matrix_PredictMultiStep := FALSE;
				RETURN;
			END_IF;
			IF PolyOrder > 1 AND pPolyTemp <> 0 THEN
				Success := HA_Matrix_PolyExpand(pLagTemp,PolyOrder,pPolyTemp);
				IF NOT Success THEN
					HA_Matrix_PredictMultiStep := FALSE;
					RETURN;
				END_IF;
				IF UseBias THEN
					Success := HA_Matrix_AddBias(pPolyTemp,pFeatTemp);
					IF NOT Success THEN
						HA_Matrix_PredictMultiStep := FALSE;
						RETURN;
					END_IF;
					Success := HA_Matrix_Predict(pFeatTemp,pBeta,pPredTemp);
				ELSE
					Success := HA_Matrix_Predict(pPolyTemp,pBeta,pPredTemp);
				END_IF;
			ELSE
				IF UseBias THEN
					Success := HA_Matrix_AddBias(pLagTemp,pFeatTemp);
					IF NOT Success THEN
						HA_Matrix_PredictMultiStep := FALSE;
						RETURN;
					END_IF;
					Success := HA_Matrix_Predict(pFeatTemp,pBeta,pPredTemp);
				ELSE
					Success := HA_Matrix_Predict(pLagTemp,pBeta,pPredTemp);
				END_IF;
			END_IF;
			IF NOT Success THEN
				HA_Matrix_PredictMultiStep := FALSE;
				RETURN;
			END_IF;
			FOR Internal.i2 := 0 TO Internal.col1-1 DO
				brsmemcpy(ADR(Internal.temp1),pPredTemp+Internal.i2*8,8);
				IF UseDerivative THEN
					brsmemcpy(ADR(Internal.temp2),pWorkState+Internal.i2*8,8);
					Internal.temp1 := Internal.temp2 + Internal.temp1;
					brsmemcpy(pWorkState+Internal.i2*8,ADR(Internal.temp1),8);
				ELSE
					brsmemcpy(pWorkState+Internal.i2*8,ADR(Internal.temp1),8);
				END_IF;
				brsmemcpy(pOut+(Internal.i1*Internal.col4+Internal.i2)*8,ADR(Internal.temp1),8);
			END_FOR;
			FOR Internal.i2 := 0 TO Internal.col1-1 DO
				brsmemcpy(ADR(Internal.temp1),pWorkState+Internal.i2*8,8);
				Success := HA_Matrix_RollingUpdate(pWorkHist,Internal.temp1);
				IF NOT Success THEN
					HA_Matrix_PredictMultiStep := FALSE;
					RETURN;
				END_IF;
			END_FOR;
		END_FOR;
	END_IF;
END_FUNCTION
```

#### HA_Matrix_Ridge_Fit.st
```iecst
(* Ridge Regression Fit *)
FUNCTION HA_Matrix_Ridge_Fit
	HA_Matrix_Ridge_Fit	 			:= TRUE;
	brsmemset(ADR(Internal),0,SIZEOF(Internal));
	Internal.sizeArray				:= SIZEOF(LREAL)*(MAX_HA_MATRIX_ARRAY_IDX+1);
	Internal.sizeTotal				:= Internal.sizeArray + SIZEOF(UDINT)*2;
	brsmemcpy(ADR(Internal.row1),pX+Internal.sizeArray,4);
	brsmemcpy(ADR(Internal.col1),pX+Internal.sizeArray+4,4);
	brsmemcpy(ADR(Internal.row2),pY+Internal.sizeArray,4);
	brsmemcpy(ADR(Internal.col2),pY+Internal.sizeArray+4,4);
	IF pX = 0 OR pY = 0 OR pBeta = 0 OR pXtX = 0 OR pXtY = 0 OR pL = 0 OR Internal.row1 = 0 OR Internal.col1 = 0 OR Internal.row2 = 0 OR Internal.col2 = 0 OR Internal.row1 <> Internal.row2 OR WarmupSteps < 0 OR WarmupSteps >= Internal.row1 OR Lambda < 0.0 OR Internal.row1*Internal.col1 > MAX_HA_MATRIX_ARRAY_IDX+1 OR Internal.row2*Internal.col2 > MAX_HA_MATRIX_ARRAY_IDX+1 THEN
		HA_Matrix_Ridge_Fit	 		:= FALSE;
	ELSE
		Internal.row3 				:= Internal.row1 - WarmupSteps;
		Internal.col3 				:= Internal.col1;
		Internal.row4 				:= Internal.row2 - WarmupSteps;
		Internal.col4 				:= Internal.col2;
		IF UseBias THEN
			Internal.col3 			:= Internal.col1 + 1;
		END_IF;
		IF pXwork <> 0 THEN
			brsmemset(pXwork,0,Internal.sizeTotal);
			brsmemcpy(pXwork+Internal.sizeArray,ADR(Internal.row3),4);
			brsmemcpy(pXwork+Internal.sizeArray+4,ADR(Internal.col3),4);
			FOR Internal.i1 := WarmupSteps TO Internal.row1-1 DO
				Internal.i4 		:= Internal.i1 - WarmupSteps;
				IF UseBias THEN
					Internal.temp1 	:= 1.0;
					brsmemcpy(pXwork+(Internal.i4*Internal.col3)*8,ADR(Internal.temp1),8);
					FOR Internal.i2 := 0 TO Internal.col1-1 DO
						brsmemcpy(ADR(Internal.temp1),pX+(Internal.i1*Internal.col1+Internal.i2)*8,8);
						brsmemcpy(pXwork+(Internal.i4*Internal.col3+Internal.i2+1)*8,ADR(Internal.temp1),8);
					END_FOR;
				ELSE
					FOR Internal.i2 := 0 TO Internal.col1-1 DO
						brsmemcpy(ADR(Internal.temp1),pX+(Internal.i1*Internal.col1+Internal.i2)*8,8);
						brsmemcpy(pXwork+(Internal.i4*Internal.col3+Internal.i2)*8,ADR(Internal.temp1),8);
					END_FOR;
				END_IF;
			END_FOR;
			brsmemset(pYwork,0,Internal.sizeTotal);
			brsmemcpy(pYwork+Internal.sizeArray,ADR(Internal.row4),4);
			brsmemcpy(pYwork+Internal.sizeArray+4,ADR(Internal.col4),4);
			FOR Internal.i1 := WarmupSteps TO Internal.row2-1 DO
				Internal.i4 		:= Internal.i1 - WarmupSteps;
				FOR Internal.i2 := 0 TO Internal.col2-1 DO
					brsmemcpy(ADR(Internal.temp1),pY+(Internal.i1*Internal.col2+Internal.i2)*8,8);
					brsmemcpy(pYwork+(Internal.i4*Internal.col4+Internal.i2)*8,ADR(Internal.temp1),8);
				END_FOR;
			END_FOR;
			Success := HA_Matrix_XtX(pXwork,pXtX);
		ELSE
			Success := HA_Matrix_XtX(pX,pXtX);
		END_IF;
		IF NOT Success THEN
			HA_Matrix_Ridge_Fit 	:= FALSE;
			RETURN;
		END_IF;
		Success := HA_Matrix_AddRidge(pXtX,Lambda);
		IF NOT Success THEN
			HA_Matrix_Ridge_Fit 	:= FALSE;
			RETURN;
		END_IF;
		Success := HA_Matrix_Cholesky(pXtX,pL);
		IF NOT Success THEN
			HA_Matrix_Ridge_Fit 	:= FALSE;
			RETURN;
		END_IF;
		IF pXwork <> 0 THEN
			Success := HA_Matrix_XtY(pXwork,pYwork,pXtY);
		ELSE
			Success := HA_Matrix_XtY(pX,pY,pXtY);
		END_IF;
		IF NOT Success THEN
			HA_Matrix_Ridge_Fit 	:= FALSE;
			RETURN;
		END_IF;
		Success := HA_Matrix_CholSolve(pL,pXtY,pBeta);
		IF NOT Success THEN
			HA_Matrix_Ridge_Fit 	:= FALSE;
			RETURN;
		END_IF;
	END_IF;
END_FUNCTION
```

#### HA_Matrix_BuildLagsStride.st
```iecst
(* Build Lag Matrix with Stride *)
FUNCTION HA_Matrix_BuildLagsStride
	HA_Matrix_BuildLagsStride	 	:= TRUE;
	brsmemset(ADR(Internal),0,SIZEOF(Internal));
	Internal.sizeArray				:= SIZEOF(LREAL)*(MAX_HA_MATRIX_ARRAY_IDX+1);
	Internal.sizeTotal				:= Internal.sizeArray + SIZEOF(UDINT)*2;
	brsmemcpy(ADR(Internal.row1),pY_history+Internal.sizeArray,4);
	brsmemcpy(ADR(Internal.col1),pY_history+Internal.sizeArray+4,4);
	IF pU_history <> 0 THEN
		brsmemcpy(ADR(Internal.row2),pU_history+Internal.sizeArray,4);
		brsmemcpy(ADR(Internal.col2),pU_history+Internal.sizeArray+4,4);
	ELSE
		Internal.row2 				:= 0;
		Internal.col2 				:= 0;
	END_IF;
	IF Stride < 1 THEN
		Stride 						:= 1;
	END_IF;
	Internal.row3					:= NumOutputs*LagOrder + NumInputs*LagOrder;
	Internal.col3					:= 1;
	IF pY_history = 0 OR pOut = 0 OR LagOrder = 0 OR NumOutputs = 0 OR Internal.row1 = 0 OR Internal.col1 = 0 OR Internal.row1 < NumOutputs*LagOrder*Stride OR Internal.col1 <> 1 OR Internal.row3*Internal.col3 > MAX_HA_MATRIX_ARRAY_IDX+1 THEN
		HA_Matrix_BuildLagsStride	:= FALSE;
	ELSE
		IF pU_history <> 0 THEN
			IF NumInputs = 0 OR Internal.row2 = 0 OR Internal.col2 = 0 OR Internal.row2 < NumInputs*LagOrder*Stride OR Internal.col2 <> 1 THEN
				HA_Matrix_BuildLagsStride := FALSE;
				RETURN;
			END_IF;
		END_IF;
		brsmemset(pOut,0,Internal.sizeTotal);
		brsmemcpy(pOut+Internal.sizeArray,ADR(Internal.row3),4);
		brsmemcpy(pOut+Internal.sizeArray+4,ADR(Internal.col3),4);
		Internal.i4 				:= 0;
		FOR Internal.i1 := 0 TO LagOrder-1 DO
		    FOR Internal.i2 := 0 TO NumOutputs-1 DO
				brsmemcpy(ADR(Internal.temp1),pY_history+((Internal.i1*Stride)*NumOutputs+Internal.i2)*8,8);
				brsmemcpy(pOut+Internal.i4*8,ADR(Internal.temp1),8);
				Internal.i4 			:= Internal.i4 + 1;
		    END_FOR;
		END_FOR;
		IF pU_history <> 0 AND NumInputs > 0 THEN
			FOR Internal.i1 := 0 TO LagOrder-1 DO
			    FOR Internal.i2 := 0 TO NumInputs-1 DO
					brsmemcpy(ADR(Internal.temp1),pU_history+((Internal.i1*Stride)*NumInputs+Internal.i2)*8,8);
					brsmemcpy(pOut+Internal.i4*8,ADR(Internal.temp1),8);
					Internal.i4 		:= Internal.i4 + 1;
			    END_FOR;
			END_FOR;
		END_IF;
	END_IF;
END_FUNCTION
```

#### HA_Matrix_InitStateBuffer.st
```iecst
(* Initialize State Buffer *)
FUNCTION HA_Matrix_InitStateBuffer
	HA_Matrix_InitStateBuffer	 	:= TRUE;
	brsmemset(ADR(Internal),0,SIZEOF(Internal));
	Internal.sizeArray				:= SIZEOF(LREAL)*(MAX_HA_MATRIX_ARRAY_IDX+1);
	Internal.sizeTotal				:= Internal.sizeArray + SIZEOF(UDINT)*2;
	brsmemcpy(ADR(Internal.row1),pX+Internal.sizeArray,4);
	brsmemcpy(ADR(Internal.col1),pX+Internal.sizeArray+4,4);
	brsmemcpy(ADR(Internal.row2),pState+Internal.sizeArray,4);
	brsmemcpy(ADR(Internal.col2),pState+Internal.sizeArray+4,4);
	brsmemcpy(ADR(Internal.row3),pHistory+Internal.sizeArray,4);
	brsmemcpy(ADR(Internal.col3),pHistory+Internal.sizeArray+4,4);
	IF pX = 0 OR pState = 0 OR pHistory = 0 OR Internal.row1 = 0 OR Internal.col1 = 0 OR Internal.row2 = 0 OR Internal.col2 = 0 OR Internal.row3 = 0 OR Internal.col3 = 0 OR LagOrder < 1 OR Internal.row1 < LagOrder OR Internal.col3 <> 1 OR Internal.row2 <> 1 OR Internal.col2 <> Internal.col1 OR Internal.row3 <> LagOrder*Internal.col1 OR Internal.row1*Internal.col1 > MAX_HA_MATRIX_ARRAY_IDX+1 THEN
		HA_Matrix_InitStateBuffer	:= FALSE;
	ELSE
		FOR Internal.i2 := 0 TO Internal.col1-1 DO
			brsmemcpy(ADR(Internal.temp1),pX+((Internal.row1-1)*Internal.col1+Internal.i2)*8,8);
			brsmemcpy(pState+Internal.i2*8,ADR(Internal.temp1),8);
		END_FOR;
		FOR Internal.i1 := 0 TO LagOrder-1 DO
		    FOR Internal.i2 := 0 TO Internal.col1-1 DO
				brsmemcpy(ADR(Internal.temp1),pX+((Internal.row1-1-Internal.i1)*Internal.col1+Internal.i2)*8,8);
				brsmemcpy(pHistory+(Internal.i1*Internal.col1+Internal.i2)*8,ADR(Internal.temp1),8);
		    END_FOR;
		END_FOR;
	END_IF;
END_FUNCTION
```

#### HA_Matrix_NGRC_BuildTrainingData.st
```iecst
(* Build NGRC Training Dataset *)
FUNCTION HA_Matrix_NGRC_BuildTrainingData
	HA_Matrix_NGRC_BuildTrainingData := TRUE;
	brsmemset(ADR(Internal),0,SIZEOF(Internal));
	Internal.sizeArray				:= SIZEOF(LREAL)*(MAX_HA_MATRIX_ARRAY_IDX+1);
	Internal.sizeTotal				:= Internal.sizeArray + SIZEOF(UDINT)*2;
	brsmemcpy(ADR(Internal.row1),pX+Internal.sizeArray,4);
	brsmemcpy(ADR(Internal.col1),pX+Internal.sizeArray+4,4);
	Internal.row2					:= Internal.row1 - (LagOrder-1)*Stride - WarmupSteps;
	Internal.col2					:= Internal.col1 * LagOrder;
	IF PolyOrder = 2 THEN
		Internal.col3 				:= Internal.col2 + (Internal.col2*(Internal.col2+1))/2;
	ELSIF PolyOrder = 3 THEN
		Internal.col3 				:= Internal.col2 + (Internal.col2*(Internal.col2+1))/2 + (Internal.col2*(Internal.col2+1)*(Internal.col2+2))/6;
	ELSE
		Internal.col3 				:= Internal.col2;
	END_IF;
	Internal.row3					:= Internal.row2;
	IF UseBias THEN
		Internal.col4 				:= Internal.col3 + 1;
	ELSE
		Internal.col4 				:= Internal.col3;
	END_IF;
	Internal.row4					:= Internal.row2;
	IF pX = 0 OR pOut = 0 OR Internal.row1 = 0 OR Internal.col1 = 0 OR LagOrder < 1 OR PolyOrder < 1 OR PolyOrder > 3 OR Stride < 1 OR WarmupSteps < 0 OR Internal.row1*Internal.col1 > MAX_HA_MATRIX_ARRAY_IDX+1 OR Internal.row1 <= (LagOrder-1)*Stride + WarmupSteps OR Internal.row4*Internal.col4 > MAX_HA_MATRIX_ARRAY_IDX+1 THEN
		HA_Matrix_NGRC_BuildTrainingData := FALSE;
	ELSE
		brsmemset(pOut,0,Internal.sizeTotal);
		brsmemcpy(pOut+Internal.sizeArray,ADR(Internal.row4),4);
		brsmemcpy(pOut+Internal.sizeArray+4,ADR(Internal.col4),4);
		brsmemset(pLagWork,0,Internal.sizeTotal);
		brsmemcpy(pLagWork+Internal.sizeArray,ADR(Internal.row2),4);
		brsmemcpy(pLagWork+Internal.sizeArray+4,ADR(Internal.col2),4);
		Internal.i4 					:= 0;
		FOR Internal.i1 := WarmupSteps + (LagOrder-1)*Stride TO Internal.row1-1 DO
			FOR Internal.i2 := 0 TO LagOrder-1 DO
				Internal.row3 		:= Internal.i1 - Internal.i2*Stride;
				FOR Internal.i3 := 0 TO Internal.col1-1 DO
					brsmemcpy(ADR(Internal.temp1),pX+(Internal.row3*Internal.col1+Internal.i3)*8,8);
					brsmemcpy(pLagWork+(Internal.i4*Internal.col2+(Internal.i2*Internal.col1+Internal.i3))*8,ADR(Internal.temp1),8);
				END_FOR;
			END_FOR;
			Internal.i4 				:= Internal.i4 + 1;
		END_FOR;
		IF PolyOrder > 1 AND pPolyWork <> 0 THEN
			Success := HA_Matrix_PolyExpand(pLagWork,PolyOrder,pPolyWork);
			IF NOT Success THEN
				HA_Matrix_NGRC_BuildTrainingData := FALSE;
				RETURN;
			END_IF;
			IF UseBias THEN
				Success := HA_Matrix_AddBias(pPolyWork,pOut);
				IF NOT Success THEN
					HA_Matrix_NGRC_BuildTrainingData := FALSE;
					RETURN;
				END_IF;
			ELSE
				brsmemcpy(pOut,pPolyWork,Internal.sizeTotal);
			END_IF;
		ELSE
			IF UseBias THEN
				Success := HA_Matrix_AddBias(pLagWork,pOut);
				IF NOT Success THEN
					HA_Matrix_NGRC_BuildTrainingData := FALSE;
					RETURN;
				END_IF;
			ELSE
				brsmemcpy(pOut,pLagWork,Internal.sizeTotal);
			END_IF;
		END_IF;
	END_IF;
END_FUNCTION
```

#### HA_Matrix_NGRC_Fit.st
```iecst
(* Fit NGRC Model *)
FUNCTION HA_Matrix_NGRC_Fit
	HA_Matrix_NGRC_Fit				:= TRUE;
	brsmemset(ADR(Internal),0,SIZEOF(Internal));
	Internal.sizeArray				:= SIZEOF(LREAL)*(MAX_HA_MATRIX_ARRAY_IDX+1);
	Internal.sizeTotal				:= Internal.sizeArray + SIZEOF(UDINT)*2;
	brsmemcpy(ADR(Internal.row1),pX+Internal.sizeArray,4);
	brsmemcpy(ADR(Internal.col1),pX+Internal.sizeArray+4,4);
	brsmemcpy(ADR(Internal.row2),pY+Internal.sizeArray,4);
	brsmemcpy(ADR(Internal.col2),pY+Internal.sizeArray+4,4);
	Internal.row3					:= Internal.row1 - (LagOrder-1)*Stride - WarmupSteps;
	IF UseDerivative THEN
		Internal.row4 				:= Internal.row3 - 1;
		Internal.col4 				:= Internal.col2;
	ELSE
		Internal.row4 				:= Internal.row3;
		Internal.col4 				:= Internal.col2;
	END_IF;
	IF pX = 0 OR pY = 0 OR pBeta = 0 OR pXtX = 0 OR pXtY = 0 OR pL = 0 OR pLagWork = 0 OR pFeatWork = 0 OR Internal.row1 = 0 OR Internal.col1 = 0 OR Internal.row2 = 0 OR Internal.col2 = 0 OR LagOrder < 1 OR PolyOrder < 1 OR PolyOrder > 3 OR Stride < 1 OR WarmupSteps < 0 OR Lambda < 0.0 OR Internal.row1*Internal.col1 > MAX_HA_MATRIX_ARRAY_IDX+1 OR Internal.row2*Internal.col2 > MAX_HA_MATRIX_ARRAY_IDX+1 OR Internal.row1 <= (LagOrder-1)*Stride + WarmupSteps THEN
		HA_Matrix_NGRC_Fit			:= FALSE;
	ELSE
		Success := HA_Matrix_NGRC_BuildTrainingData(pX,LagOrder,PolyOrder,Stride,UseBias,WarmupSteps,pFeatWork,pLagWork,pPolyWork);
		IF NOT Success THEN
			HA_Matrix_NGRC_Fit		:= FALSE;
			RETURN;
		END_IF;
		IF UseDerivative THEN
			(* Adjust feature matrix dimensions to match derivative targets *)
			brsmemcpy(pFeatWork+Internal.sizeArray,ADR(Internal.row4),4);

			(* Build derivative targets *)
			brsmemset(pYwork,0,Internal.sizeTotal);
			brsmemcpy(pYwork+Internal.sizeArray,ADR(Internal.row4),4);
			brsmemcpy(pYwork+Internal.sizeArray+4,ADR(Internal.col4),4);
			FOR Internal.i1 := WarmupSteps + (LagOrder-1)*Stride TO Internal.row1-2 DO
				Internal.i4 		:= Internal.i1 - WarmupSteps - (LagOrder-1)*Stride;
				FOR Internal.i2 := 0 TO Internal.col1-1 DO
					brsmemcpy(ADR(Internal.temp1),pX+((Internal.i1+1)*Internal.col1+Internal.i2)*8,8);
					brsmemcpy(ADR(Internal.temp2),pX+(Internal.i1*Internal.col1+Internal.i2)*8,8);
					Internal.temp3 	:= Internal.temp1 - Internal.temp2;
					brsmemcpy(pYwork+(Internal.i4*Internal.col4+Internal.i2)*8,ADR(Internal.temp3),8);
				END_FOR;
			END_FOR;
			Success := HA_Matrix_XtX(pFeatWork,pXtX);
			IF NOT Success THEN
				HA_Matrix_NGRC_Fit	:= FALSE;
				RETURN;
			END_IF;
			Success := HA_Matrix_AddRidge(pXtX,Lambda);
			IF NOT Success THEN
				HA_Matrix_NGRC_Fit	:= FALSE;
				RETURN;
			END_IF;
			Success := HA_Matrix_Cholesky(pXtX,pL);
			IF NOT Success THEN
				HA_Matrix_NGRC_Fit	:= FALSE;
				RETURN;
			END_IF;
			Success := HA_Matrix_XtY(pFeatWork,pYwork,pXtY);
			IF NOT Success THEN
				HA_Matrix_NGRC_Fit	:= FALSE;
				RETURN;
			END_IF;
			Success := HA_Matrix_CholSolve(pL,pXtY,pBeta);
			IF NOT Success THEN
				HA_Matrix_NGRC_Fit	:= FALSE;
				RETURN;
			END_IF;
		ELSE
			brsmemset(pYwork,0,Internal.sizeTotal);
			brsmemcpy(pYwork+Internal.sizeArray,ADR(Internal.row4),4);
			brsmemcpy(pYwork+Internal.sizeArray+4,ADR(Internal.col4),4);
			FOR Internal.i1 := WarmupSteps + (LagOrder-1)*Stride TO Internal.row1-1 DO
				Internal.i4 		:= Internal.i1 - WarmupSteps - (LagOrder-1)*Stride;
				FOR Internal.i2 := 0 TO Internal.col2-1 DO
					brsmemcpy(ADR(Internal.temp1),pY+(Internal.i1*Internal.col2+Internal.i2)*8,8);
					brsmemcpy(pYwork+(Internal.i4*Internal.col4+Internal.i2)*8,ADR(Internal.temp1),8);
				END_FOR;
			END_FOR;
			Success := HA_Matrix_XtX(pFeatWork,pXtX);
			IF NOT Success THEN
				HA_Matrix_NGRC_Fit	:= FALSE;
				RETURN;
			END_IF;
			Success := HA_Matrix_AddRidge(pXtX,Lambda);
			IF NOT Success THEN
				HA_Matrix_NGRC_Fit	:= FALSE;
				RETURN;
			END_IF;
			Success := HA_Matrix_Cholesky(pXtX,pL);
			IF NOT Success THEN
				HA_Matrix_NGRC_Fit	:= FALSE;
				RETURN;
			END_IF;
			Success := HA_Matrix_XtY(pFeatWork,pYwork,pXtY);
			IF NOT Success THEN
				HA_Matrix_NGRC_Fit	:= FALSE;
				RETURN;
			END_IF;
			Success := HA_Matrix_CholSolve(pL,pXtY,pBeta);
			IF NOT Success THEN
				HA_Matrix_NGRC_Fit	:= FALSE;
				RETURN;
			END_IF;
		END_IF;
	END_IF;
END_FUNCTION
```

#### HA_Matrix_NGRC_InitState.st
```iecst
(* Initialize NGRC State Buffer *)
FUNCTION HA_Matrix_NGRC_InitState
	HA_Matrix_NGRC_InitState		:= TRUE;
	brsmemset(ADR(Internal),0,SIZEOF(Internal));
	Internal.sizeArray				:= SIZEOF(LREAL)*(MAX_HA_MATRIX_ARRAY_IDX+1);
	Internal.sizeTotal				:= Internal.sizeArray + SIZEOF(UDINT)*2;

	(* Read INPUT dimensions *)
	brsmemcpy(ADR(Internal.row1),pX+Internal.sizeArray,4);
	brsmemcpy(ADR(Internal.col1),pX+Internal.sizeArray+4,4);

	(* Validate INPUTS only - removed output dimension validation *)
	IF pX = 0 OR pState = 0 OR pHistory = 0 OR
	   Internal.row1 = 0 OR Internal.col1 = 0 OR
	   LagOrder < 1 OR Stride < 1 OR
	   Internal.row1 < (LagOrder-1)*Stride + 1 OR
	   Internal.row1*Internal.col1 > MAX_HA_MATRIX_ARRAY_IDX+1 THEN
		HA_Matrix_NGRC_InitState	:= FALSE;
		RETURN;
	END_IF;

	(* CALCULATE output dimensions *)
	Internal.row2					:= 1;                    (* State: 1 row *)
	Internal.col2					:= Internal.col1;        (* State: same cols as input *)
	Internal.row3					:= LagOrder*Internal.col1; (* History: LagOrder*cols rows *)
	Internal.col3					:= 1;                    (* History: 1 column *)

	(* Verify output will fit in array *)
	IF Internal.row2*Internal.col2 > MAX_HA_MATRIX_ARRAY_IDX+1 OR
	   Internal.row3*Internal.col3 > MAX_HA_MATRIX_ARRAY_IDX+1 THEN
		HA_Matrix_NGRC_InitState	:= FALSE;
		RETURN;
	END_IF;

	(* INITIALIZE State array *)
	brsmemset(pState,0,Internal.sizeTotal);
	brsmemcpy(pState+Internal.sizeArray,ADR(Internal.row2),4);
	brsmemcpy(pState+Internal.sizeArray+4,ADR(Internal.col2),4);

	(* INITIALIZE History array *)
	brsmemset(pHistory,0,Internal.sizeTotal);
	brsmemcpy(pHistory+Internal.sizeArray,ADR(Internal.row3),4);
	brsmemcpy(pHistory+Internal.sizeArray+4,ADR(Internal.col3),4);

	(* POPULATE State with last sample from X *)
	FOR Internal.i2 := 0 TO Internal.col1-1 DO
		brsmemcpy(ADR(Internal.temp1),pX+((Internal.row1-1)*Internal.col1+Internal.i2)*8,8);
		brsmemcpy(pState+Internal.i2*8,ADR(Internal.temp1),8);
	END_FOR;

	(* POPULATE History with last LagOrder samples at stride intervals *)
	FOR Internal.i1 := 0 TO LagOrder-1 DO
	    FOR Internal.i2 := 0 TO Internal.col1-1 DO
			Internal.row4 		:= Internal.row1-1-Internal.i1*Stride;
			brsmemcpy(ADR(Internal.temp1),pX+(Internal.row4*Internal.col1+Internal.i2)*8,8);
			brsmemcpy(pHistory+(Internal.i1*Internal.col1+Internal.i2)*8,ADR(Internal.temp1),8);
	    END_FOR;
	END_FOR;
END_FUNCTION
```

#### HA_Matrix_NGRC_Predict.st
```iecst
(* NGRC Single-Step Prediction *)
FUNCTION HA_Matrix_NGRC_Predict
	HA_Matrix_NGRC_Predict			:= TRUE;
	brsmemset(ADR(Internal),0,SIZEOF(Internal));
	Internal.sizeArray				:= SIZEOF(LREAL)*(MAX_HA_MATRIX_ARRAY_IDX+1);
	Internal.sizeTotal				:= Internal.sizeArray + SIZEOF(UDINT)*2;
	brsmemcpy(ADR(Internal.row1),pHistory+Internal.sizeArray,4);
	brsmemcpy(ADR(Internal.col1),pHistory+Internal.sizeArray+4,4);
	brsmemcpy(ADR(Internal.row2),pBeta+Internal.sizeArray,4);
	brsmemcpy(ADR(Internal.col2),pBeta+Internal.sizeArray+4,4);
	Internal.row3					:= Internal.col1;
	Internal.col3					:= 1;
	IF pHistory = 0 OR pBeta = 0 OR pOut = 0 OR pLagWork = 0 OR Internal.row1 = 0 OR Internal.col1 = 0 OR Internal.row2 = 0 OR Internal.col2 = 0 OR LagOrder < 1 OR PolyOrder < 1 OR PolyOrder > 3 OR Internal.row1*Internal.col1 > MAX_HA_MATRIX_ARRAY_IDX+1 OR Internal.row2*Internal.col2 > MAX_HA_MATRIX_ARRAY_IDX+1 THEN
		HA_Matrix_NGRC_Predict		:= FALSE;
	ELSE
		brsmemset(pLagWork,0,Internal.sizeTotal);
		brsmemcpy(pLagWork+Internal.sizeArray,ADR(Internal.row3),4);
		brsmemcpy(pLagWork+Internal.sizeArray+4,ADR(Internal.col3),4);
		FOR Internal.i1 := 0 TO Internal.row1-1 DO
			brsmemcpy(ADR(Internal.temp1),pHistory+Internal.i1*8,8);
			brsmemcpy(pLagWork+Internal.i1*8,ADR(Internal.temp1),8);
		END_FOR;
		IF PolyOrder > 1 AND pPolyWork <> 0 THEN
			Success := HA_Matrix_PolyExpand(pLagWork,PolyOrder,pPolyWork);
			IF NOT Success THEN
				HA_Matrix_NGRC_Predict := FALSE;
				RETURN;
			END_IF;
			IF UseBias THEN
				Success := HA_Matrix_AddBias(pPolyWork,pFeatWork);
				IF NOT Success THEN
					HA_Matrix_NGRC_Predict := FALSE;
					RETURN;
				END_IF;
				Success := HA_Matrix_Predict(pFeatWork,pBeta,pOut);
			ELSE
				Success := HA_Matrix_Predict(pPolyWork,pBeta,pOut);
			END_IF;
		ELSE
			IF UseBias THEN
				Success := HA_Matrix_AddBias(pLagWork,pFeatWork);
				IF NOT Success THEN
					HA_Matrix_NGRC_Predict := FALSE;
					RETURN;
				END_IF;
				Success := HA_Matrix_Predict(pFeatWork,pBeta,pOut);
			ELSE
				Success := HA_Matrix_Predict(pLagWork,pBeta,pOut);
			END_IF;
		END_IF;
		IF NOT Success THEN
			HA_Matrix_NGRC_Predict	:= FALSE;
			RETURN;
		END_IF;
	END_IF;
END_FUNCTION
```

#### HA_Matrix_NGRC_PredictMultiStep.st
```iecst
(* NGRC Multi-Step Prediction *)
FUNCTION HA_Matrix_NGRC_PredictMultiStep
	HA_Matrix_NGRC_PredictMultiStep	:= TRUE;
	brsmemset(ADR(Internal),0,SIZEOF(Internal));
	Internal.sizeArray				:= SIZEOF(LREAL)*(MAX_HA_MATRIX_ARRAY_IDX+1);
	Internal.sizeTotal				:= Internal.sizeArray + SIZEOF(UDINT)*2;
	brsmemcpy(ADR(Internal.row1),pState+Internal.sizeArray,4);
	brsmemcpy(ADR(Internal.col1),pState+Internal.sizeArray+4,4);
	brsmemcpy(ADR(Internal.row2),pBeta+Internal.sizeArray,4);
	brsmemcpy(ADR(Internal.col2),pBeta+Internal.sizeArray+4,4);
	brsmemcpy(ADR(Internal.row3),pHistory+Internal.sizeArray,4);
	brsmemcpy(ADR(Internal.col3),pHistory+Internal.sizeArray+4,4);
	Internal.row4					:= Steps;
	Internal.col4					:= Internal.col1;
	IF pState = 0 OR pBeta = 0 OR pHistory = 0 OR pOut = 0 OR pLagWork = 0 OR pPredWork = 0 OR pWorkState = 0 OR pWorkHist = 0 OR Internal.row1 = 0 OR Internal.col1 = 0 OR Internal.row2 = 0 OR Internal.col2 = 0 OR Internal.row3 = 0 OR Internal.col3 = 0 OR Steps <= 0 OR LagOrder < 1 OR PolyOrder < 1 OR PolyOrder > 3 OR Stride < 1 OR Internal.row1 <> 1 OR Internal.col3 <> 1 OR Internal.col2 <> Internal.col1 OR Internal.row4*Internal.col4 > MAX_HA_MATRIX_ARRAY_IDX+1 THEN
		HA_Matrix_NGRC_PredictMultiStep := FALSE;
	ELSE
		brsmemset(pOut,0,Internal.sizeTotal);
		brsmemcpy(pOut+Internal.sizeArray,ADR(Internal.row4),4);
		brsmemcpy(pOut+Internal.sizeArray+4,ADR(Internal.col4),4);
		FOR Internal.i1 := 0 TO Internal.col1-1 DO
			brsmemcpy(ADR(Internal.temp1),pState+Internal.i1*8,8);
			brsmemcpy(pWorkState+Internal.i1*8,ADR(Internal.temp1),8);
		END_FOR;
		FOR Internal.i1 := 0 TO Internal.row3-1 DO
			brsmemcpy(ADR(Internal.temp1),pHistory+Internal.i1*8,8);
			brsmemcpy(pWorkHist+Internal.i1*8,ADR(Internal.temp1),8);
		END_FOR;
		FOR Internal.i1 := 0 TO Steps-1 DO
			Success := HA_Matrix_NGRC_Predict(pWorkHist,pBeta,LagOrder,PolyOrder,UseBias,pPredWork,pLagWork,pPolyWork,pFeatWork);
			IF NOT Success THEN
				HA_Matrix_NGRC_PredictMultiStep := FALSE;
				RETURN;
			END_IF;
			FOR Internal.i2 := 0 TO Internal.col1-1 DO
				brsmemcpy(ADR(Internal.temp1),pPredWork+Internal.i2*8,8);
				IF UseDerivative THEN
					brsmemcpy(ADR(Internal.temp2),pWorkState+Internal.i2*8,8);
					Internal.temp1 := Internal.temp2 + Internal.temp1;
					brsmemcpy(pWorkState+Internal.i2*8,ADR(Internal.temp1),8);
				ELSE
					brsmemcpy(pWorkState+Internal.i2*8,ADR(Internal.temp1),8);
				END_IF;
				brsmemcpy(pOut+(Internal.i1*Internal.col4+Internal.i2)*8,ADR(Internal.temp1),8);
			END_FOR;
			FOR Internal.i2 := Internal.row3-1 TO Internal.col1 BY -1 DO
			    brsmemcpy(ADR(Internal.temp1),pWorkHist+(Internal.i2-Internal.col1)*8,8);
			    brsmemcpy(pWorkHist+Internal.i2*8,ADR(Internal.temp1),8);
			END_FOR;
			FOR Internal.i2 := 0 TO Internal.col1-1 DO
				brsmemcpy(ADR(Internal.temp1),pWorkState+Internal.i2*8,8);
				brsmemcpy(pWorkHist+Internal.i2*8,ADR(Internal.temp1),8);
			END_FOR;
		END_FOR;
	END_IF;
END_FUNCTION
```

#### FB_NGRC.st
```iecst
FUNCTION_BLOCK FB_NGRC

IF NOT Enable THEN
	Status := NGRC_IDLE;
	Error := NGRC_ERR_NONE;
	Ready := FALSE;
	Busy := FALSE;
	Done := FALSE;
	IsTrained := FALSE;
	RETURN;
END_IF;

IF Reset AND NOT ResetTrigger THEN
	ResetTrigger := TRUE;
	Status := NGRC_IDLE;
	Error := NGRC_ERR_NONE;
	Done := FALSE;
	IsTrained := FALSE;
	Internal.TrainStep := 0;
	brsmemset(ADR(Internal),0,SIZEOF(Internal));
END_IF;
IF NOT Reset THEN
	ResetTrigger := FALSE;
END_IF;

Ready := (Status = NGRC_IDLE OR Status = NGRC_TRAINED) AND NOT Busy;
Busy := (Status = NGRC_TRAINING OR Status = NGRC_PREDICTING);

IF Train AND NOT TrainTrigger AND NOT Busy THEN
	TrainTrigger := TRUE;
	Done := FALSE;
	Status := NGRC_TRAINING;
	Error := NGRC_ERR_NONE;
	Internal.TrainStep := 0;
	StartTime := 0;
END_IF;
IF NOT Train THEN
	TrainTrigger := FALSE;
END_IF;

IF Predict AND NOT PredictTrigger AND NOT Busy THEN
	PredictTrigger := TRUE;
	Done := FALSE;
	IF NOT IsTrained THEN
		Status := NGRC_ERROR;
		Error := NGRC_ERR_NOT_TRAINED;
		Done := TRUE;
	ELSE
		Status := NGRC_PREDICTING;
		Error := NGRC_ERR_NONE;
		StartTime := 0;
	END_IF;
END_IF;
IF NOT Predict THEN
	PredictTrigger := FALSE;
END_IF;

CASE Status OF
	NGRC_IDLE:
		;

	NGRC_TRAINING:
		IF Internal.TrainStep = 0 THEN
			NumDims := TrainingData.Col;
			NumSamples := TrainingData.Row;
			IF NumDims = 0 OR NumSamples = 0 THEN
				Status := NGRC_ERROR;
				Error := NGRC_ERR_NO_DATA;
				Done := TRUE;
				RETURN;
			END_IF;
			IF Config.LagOrder < 1 OR Config.PolyOrder < 1 OR Config.PolyOrder > 3 OR Config.Stride < 1 OR Config.Lambda < 0.0 THEN
				Status := NGRC_ERROR;
				Error := NGRC_ERR_INVALID_CONFIG;
				Done := TRUE;
				RETURN;
			END_IF;
			IF NumSamples <= (Config.LagOrder-1)*Config.Stride + Config.WarmupSteps + 1 THEN
				Status := NGRC_ERROR;
				Error := NGRC_ERR_INSUFFICIENT_DATA;
				Done := TRUE;
				RETURN;
			END_IF;
			Stats.NumSamples := NumSamples - (Config.LagOrder-1)*Config.Stride - Config.WarmupSteps;
			IF Config.PolyOrder = 2 THEN
				Stats.NumFeatures := NumDims*Config.LagOrder + (NumDims*Config.LagOrder*(NumDims*Config.LagOrder+1))/2;
			ELSIF Config.PolyOrder = 3 THEN
				Stats.NumFeatures := NumDims*Config.LagOrder + (NumDims*Config.LagOrder*(NumDims*Config.LagOrder+1))/2 + (NumDims*Config.LagOrder*(NumDims*Config.LagOrder+1)*(NumDims*Config.LagOrder+2))/6;
			ELSE
				Stats.NumFeatures := NumDims*Config.LagOrder;
			END_IF;
			IF Config.UseBias THEN
				Stats.NumFeatures := Stats.NumFeatures + 1;
			END_IF;
			IF Stats.NumFeatures*Stats.NumFeatures > MAX_HA_MATRIX_ARRAY_IDX+1 THEN
				Status := NGRC_ERROR;
				Error := NGRC_ERR_MEMORY;
				Done := TRUE;
				RETURN;
			END_IF;
			Internal.TrainStep := 1;

		ELSIF Internal.TrainStep = 1 THEN
			Success := HA_Matrix_NGRC_Fit(
				ADR(TrainingData),
				ADR(TrainingData),
				Config.LagOrder,
				Config.PolyOrder,
				Config.Stride,
				Config.Lambda,
				Config.UseBias,
				Config.UseDerivative,
				Config.WarmupSteps,
				ADR(Internal.Beta),
				ADR(Internal.XtX),
				ADR(Internal.XtY),
				ADR(Internal.L),
				ADR(Internal.LagWork),
				ADR(Internal.PolyWork),
				ADR(Internal.FeatWork),
				ADR(Internal.Ywork)
			);
			IF NOT Success THEN
				Status := NGRC_ERROR;
				Error := NGRC_ERR_TRAINING_FAILED;
				Done := TRUE;
				RETURN;
			END_IF;
			Internal.TrainStep := 2;

		ELSIF Internal.TrainStep = 2 THEN
			Success := HA_Matrix_NGRC_InitState(
				ADR(TrainingData),
				Config.LagOrder,
				Config.Stride,
				ADR(Internal.State),
				ADR(Internal.History)
			);
			IF NOT Success THEN
				Status := NGRC_ERROR;
				Error := NGRC_ERR_TRAINING_FAILED;
				Done := TRUE;
				RETURN;
			END_IF;
			Internal.TrainStep := 3;

		ELSIF Internal.TrainStep = 3 THEN
			IsTrained := TRUE;
			Status := NGRC_TRAINED;
			Done := TRUE;
			Internal.TrainStep := 0;
		END_IF;

	NGRC_TRAINED:
		;

	NGRC_PREDICTING:
		IF PredictSteps <= 0 THEN
			PredictSteps := 1;
		END_IF;
		Success := HA_Matrix_NGRC_PredictMultiStep(
			ADR(Internal.State),
			ADR(Internal.Beta),
			ADR(Internal.History),
			PredictSteps,
			Config.LagOrder,
			Config.PolyOrder,
			Config.Stride,
			Config.UseBias,
			Config.UseDerivative,
			ADR(PredictionOutput),
			ADR(Internal.LagWork),
			ADR(Internal.PolyWork),
			ADR(Internal.FeatWork),
			ADR(Internal.PredWork),
			ADR(Internal.WorkState),
			ADR(Internal.WorkHist)
		);
		IF NOT Success THEN
			Status := NGRC_ERROR;
			Error := NGRC_ERR_PREDICTION_FAILED;
			Done := TRUE;
		ELSE
			Status := NGRC_TRAINED;
			Done := TRUE;
		END_IF;

	NGRC_ERROR:
		;

END_CASE;

END_FUNCTION_BLOCK
```
